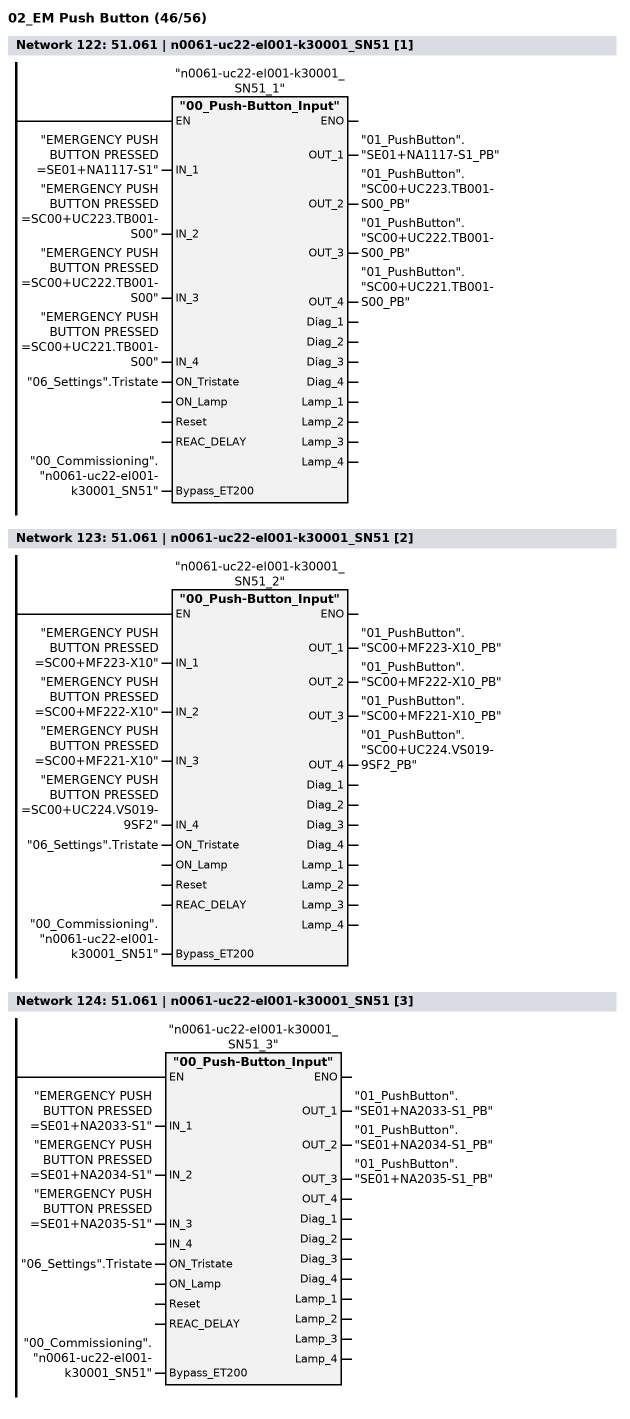
   RUNG wire#powerrail
      "n0061-uc22-el001-k30001_SN51_1"(IN_1 := "EMERGENCY PUSH BUTTON PRESSED =SE01+NA1117-S1", IN_2 := "EMERGENCY PUSH BUTTON PRESSED =SC00+UC223.TB001-S00", IN_3 := "EMERGENCY PUSH BUTTON PRESSED =SC00+UC222.TB001-S00", IN_4 := "EMERGENCY PUSH BUTTON PRESSED =SC00+UC221.TB001-S00", ON_Tristate := "06_Settings".Tristate, ON_Lamp :=, Reset :=, REAC_DELAY :=, Bypass_ET200 := "00_Commissioning"."n0061-uc22-el001-k30001_SN51", OUT_1 => "01_PushButton"."SE01+NA1117-S1_PB", OUT_2 => "01_PushButton"."SC00+UC223.TB001-S00_PB", OUT_3 => "01_PushButton"."SC00+UC222.TB001-S00_PB", OUT_4 => "01_PushButton"."SC00+UC221.TB001-S00_PB", Diag_1 =>, Diag_2 =>, Diag_3 =>, Diag_4 =>, Lamp_1 =>, Lamp_2 =>, Lamp_3 =>, Lamp_4 =>)
   END_RUNG
   // the same network as SCL:
   "n0061-uc22-el001-k30001_SN51_1"(IN_1 := "EMERGENCY PUSH BUTTON PRESSED =SE01+NA1117-S1",   // "00_Push-Button_Input"
                           IN_2 := "EMERGENCY PUSH BUTTON PRESSED =SC00+UC223.TB001-S00",
                           IN_3 := "EMERGENCY PUSH BUTTON PRESSED =SC00+UC222.TB001-S00",
                           IN_4 := "EMERGENCY PUSH BUTTON PRESSED =SC00+UC221.TB001-S00",
                           ON_Tristate := "06_Settings".Tristate,
                           Bypass_ET200 := "00_Commissioning"."n0061-uc22-el001-k30001_SN51",
                           OUT_1 => "01_PushButton"."SE01+NA1117-S1_PB",
                           OUT_2 => "01_PushButton"."SC00+UC223.TB001-S00_PB",
                           OUT_3 => "01_PushButton"."SC00+UC222.TB001-S00_PB",
                           OUT_4 => "01_PushButton"."SC00+UC221.TB001-S00_PB");
END_REGION

REGION Network 123: 51.061 | n0061-uc22-el001-k30001_SN51 [2]
   RUNG wire#powerrail
      "n0061-uc22-el001-k30001_SN51_2"(IN_1 := "EMERGENCY PUSH BUTTON PRESSED =SC00+MF223-X10", IN_2 := "EMERGENCY PUSH BUTTON PRESSED =SC00+MF222-X10", IN_3 := "EMERGENCY PUSH BUTTON PRESSED =SC00+MF221-X10", IN_4 := "EMERGENCY PUSH BUTTON PRESSED =SC00+UC224.VS019-9SF2", ON_Tristate := "06_Settings".Tristate, ON_Lamp :=, Reset :=, REAC_DELAY :=, Bypass_ET200 := "00_Commissioning"."n0061-uc22-el001-k30001_SN51", OUT_1 => "01_PushButton"."SC00+MF223-X10_PB", OUT_2 => "01_PushButton"."SC00+MF222-X10_PB", OUT_3 => "01_PushButton"."SC00+MF221-X10_PB", OUT_4 => "01_PushButton"."SC00+UC224.VS019-9SF2_PB", Diag_1 =>, Diag_2 =>, Diag_3 =>, Diag_4 =>, Lamp_1 =>, Lamp_2 =>, Lamp_3 =>, Lamp_4 =>)
   END_RUNG
   // the same network as SCL:
   "n0061-uc22-el001-k30001_SN51_2"(IN_1 := "EMERGENCY PUSH BUTTON PRESSED =SC00+MF223-X10",   // "00_Push-Button_Input"
                           IN_2 := "EMERGENCY PUSH BUTTON PRESSED =SC00+MF222-X10",
                           IN_3 := "EMERGENCY PUSH BUTTON PRESSED =SC00+MF221-X10",
                           IN_4 := "EMERGENCY PUSH BUTTON PRESSED =SC00+UC224.VS019-9SF2",
                           ON_Tristate := "06_Settings".Tristate,
                           Bypass_ET200 := "00_Commissioning"."n0061-uc22-el001-k30001_SN51",
                           OUT_1 => "01_PushButton"."SC00+MF223-X10_PB",
                           OUT_2 => "01_PushButton"."SC00+MF222-X10_PB",
                           OUT_3 => "01_PushButton"."SC00+MF221-X10_PB",
                           OUT_4 => "01_PushButton"."SC00+UC224.VS019-9SF2_PB");
END_REGION

REGION Network 124: 51.061 | n0061-uc22-el001-k30001_SN51 [3]
   RUNG wire#powerrail
      "n0061-uc22-el001-k30001_SN51_3"(IN_1 := "EMERGENCY PUSH BUTTON PRESSED =SE01+NA2033-S1", IN_2 := "EMERGENCY PUSH BUTTON PRESSED =SE01+NA2034-S1", IN_3 := "EMERGENCY PUSH BUTTON PRESSED =SE01+NA2035-S1", IN_4 :=, ON_Tristate := "06_Settings".Tristate, ON_Lamp :=, Reset :=, REAC_DELAY :=, Bypass_ET200 := "00_Commissioning"."n0061-uc22-el001-k30001_SN51", OUT_1 => "01_PushButton"."SE01+NA2033-S1_PB", OUT_2 => "01_PushButton"."SE01+NA2034-S1_PB", OUT_3 => "01_PushButton"."SE01+NA2035-S1_PB", OUT_4 =>, Diag_1 =>, Diag_2 =>, Diag_3 =>, Diag_4 =>, Lamp_1 =>, Lamp_2 =>, Lamp_3 =>, Lamp_4 =>)
   END_RUNG
   // the same network as SCL:
   "n0061-uc22-el001-k30001_SN51_3"(IN_1 := "EMERGENCY PUSH BUTTON PRESSED =SE01+NA2033-S1",   // "00_Push-Button_Input"
                           IN_2 := "EMERGENCY PUSH BUTTON PRESSED =SE01+NA2034-S1",
                           IN_3 := "EMERGENCY PUSH BUTTON PRESSED =SE01+NA2035-S1",
                           ON_Tristate := "06_Settings".Tristate,
                           Bypass_ET200 := "00_Commissioning"."n0061-uc22-el001-k30001_SN51",
                           OUT_1 => "01_PushButton"."SE01+NA2033-S1_PB",
                           OUT_2 => "01_PushButton"."SE01+NA2034-S1_PB",
                           OUT_3 => "01_PushButton"."SE01+NA2035-S1_PB");
END_REGION

REGION Network 125: 51.062 | n0062-uc224-xn10_SN51 [1]
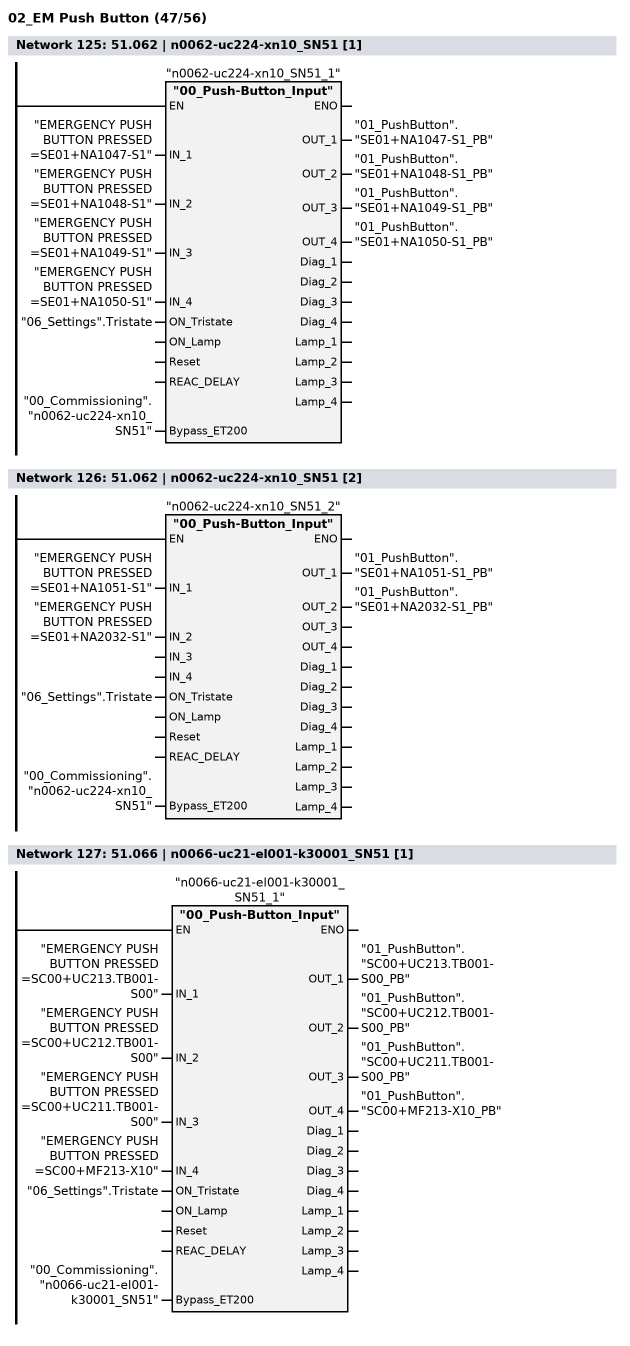
   RUNG wire#powerrail
      "n0062-uc224-xn10_SN51_1"(IN_1 := "EMERGENCY PUSH BUTTON PRESSED =SE01+NA1047-S1", IN_2 := "EMERGENCY PUSH BUTTON PRESSED =SE01+NA1048-S1", IN_3 := "EMERGENCY PUSH BUTTON PRESSED =SE01+NA1049-S1", IN_4 := "EMERGENCY PUSH BUTTON PRESSED =SE01+NA1050-S1", ON_Tristate := "06_Settings".Tristate, ON_Lamp :=, Reset :=, REAC_DELAY :=, Bypass_ET200 := "00_Commissioning"."n0062-uc224-xn10_SN51", OUT_1 => "01_PushButton"."SE01+NA1047-S1_PB", OUT_2 => "01_PushButton"."SE01+NA1048-S1_PB", OUT_3 => "01_PushButton"."SE01+NA1049-S1_PB", OUT_4 => "01_PushButton"."SE01+NA1050-S1_PB", Diag_1 =>, Diag_2 =>, Diag_3 =>, Diag_4 =>, Lamp_1 =>, Lamp_2 =>, Lamp_3 =>, Lamp_4 =>)
   END_RUNG
   // the same network as SCL:
   "n0062-uc224-xn10_SN51_1"(IN_1 := "EMERGENCY PUSH BUTTON PRESSED =SE01+NA1047-S1",   // "00_Push-Button_Input"
                           IN_2 := "EMERGENCY PUSH BUTTON PRESSED =SE01+NA1048-S1",
                           IN_3 := "EMERGENCY PUSH BUTTON PRESSED =SE01+NA1049-S1",
                           IN_4 := "EMERGENCY PUSH BUTTON PRESSED =SE01+NA1050-S1",
                           ON_Tristate := "06_Settings".Tristate,
                           Bypass_ET200 := "00_Commissioning"."n0062-uc224-xn10_SN51",
                           OUT_1 => "01_PushButton"."SE01+NA1047-S1_PB",
                           OUT_2 => "01_PushButton"."SE01+NA1048-S1_PB",
                           OUT_3 => "01_PushButton"."SE01+NA1049-S1_PB",
                           OUT_4 => "01_PushButton"."SE01+NA1050-S1_PB");
END_REGION

REGION Network 126: 51.062 | n0062-uc224-xn10_SN51 [2]
   RUNG wire#powerrail
      "n0062-uc224-xn10_SN51_2"(IN_1 := "EMERGENCY PUSH BUTTON PRESSED =SE01+NA1051-S1", IN_2 := "EMERGENCY PUSH BUTTON PRESSED =SE01+NA2032-S1", IN_3 :=, IN_4 :=, ON_Tristate := "06_Settings".Tristate, ON_Lamp :=, Reset :=, REAC_DELAY :=, Bypass_ET200 := "00_Commissioning"."n0062-uc224-xn10_SN51", OUT_1 => "01_PushButton"."SE01+NA1051-S1_PB", OUT_2 => "01_PushButton"."SE01+NA2032-S1_PB", OUT_3 =>, OUT_4 =>, Diag_1 =>, Diag_2 =>, Diag_3 =>, Diag_4 =>, Lamp_1 =>, Lamp_2 =>, Lamp_3 =>, Lamp_4 =>)
   END_RUNG
   // the same network as SCL:
   "n0062-uc224-xn10_SN51_2"(IN_1 := "EMERGENCY PUSH BUTTON PRESSED =SE01+NA1051-S1",   // "00_Push-Button_Input"
                           IN_2 := "EMERGENCY PUSH BUTTON PRESSED =SE01+NA2032-S1",
                           ON_Tristate := "06_Settings".Tristate,
                           Bypass_ET200 := "00_Commissioning"."n0062-uc224-xn10_SN51",
                           OUT_1 => "01_PushButton"."SE01+NA1051-S1_PB",
                           OUT_2 => "01_PushButton"."SE01+NA2032-S1_PB");
END_REGION

REGION Network 127: 51.066 | n0066-uc21-el001-k30001_SN51 [1]
   RUNG wire#powerrail
      "n0066-uc21-el001-k30001_SN51_1"(IN_1 := "EMERGENCY PUSH BUTTON PRESSED =SC00+UC213.TB001-S00", IN_2 := "EMERGENCY PUSH BUTTON PRESSED =SC00+UC212.TB001-S00", IN_3 := "EMERGENCY PUSH BUTTON PRESSED =SC00+UC211.TB001-S00", IN_4 := "EMERGENCY PUSH BUTTON PRESSED =SC00+MF213-X10", ON_Tristate := "06_Settings".Tristate, ON_Lamp :=, Reset :=, REAC_DELAY :=, Bypass_ET200 := "00_Commissioning"."n0066-uc21-el001-k30001_SN51", OUT_1 => "01_PushButton"."SC00+UC213.TB001-S00_PB", OUT_2 => "01_PushButton"."SC00+UC212.TB001-S00_PB", OUT_3 => "01_PushButton"."SC00+UC211.TB001-S00_PB", OUT_4 => "01_PushButton"."SC00+MF213-X10_PB", Diag_1 =>, Diag_2 =>, Diag_3 =>, Diag_4 =>, Lamp_1 =>, Lamp_2 =>, Lamp_3 =>, Lamp_4 =>)
   END_RUNG
   // the same network as SCL:
   "n0066-uc21-el001-k30001_SN51_1"(IN_1 := "EMERGENCY PUSH BUTTON PRESSED =SC00+UC213.TB001-S00",   // "00_Push-Button_Input"
                           IN_2 := "EMERGENCY PUSH BUTTON PRESSED =SC00+UC212.TB001-S00",
                           IN_3 := "EMERGENCY PUSH BUTTON PRESSED =SC00+UC211.TB001-S00",
                           IN_4 := "EMERGENCY PUSH BUTTON PRESSED =SC00+MF213-X10",
                           ON_Tristate := "06_Settings".Tristate,
                           Bypass_ET200 := "00_Commissioning"."n0066-uc21-el001-k30001_SN51",
                           OUT_1 => "01_PushButton"."SC00+UC213.TB001-S00_PB",
                           OUT_2 => "01_PushButton"."SC00+UC212.TB001-S00_PB",
                           OUT_3 => "01_PushButton"."SC00+UC211.TB001-S00_PB",
                           OUT_4 => "01_PushButton"."SC00+MF213-X10_PB");
END_REGION

REGION Network 128: 51.066 | n0066-uc21-el001-k30001_SN51 [2]
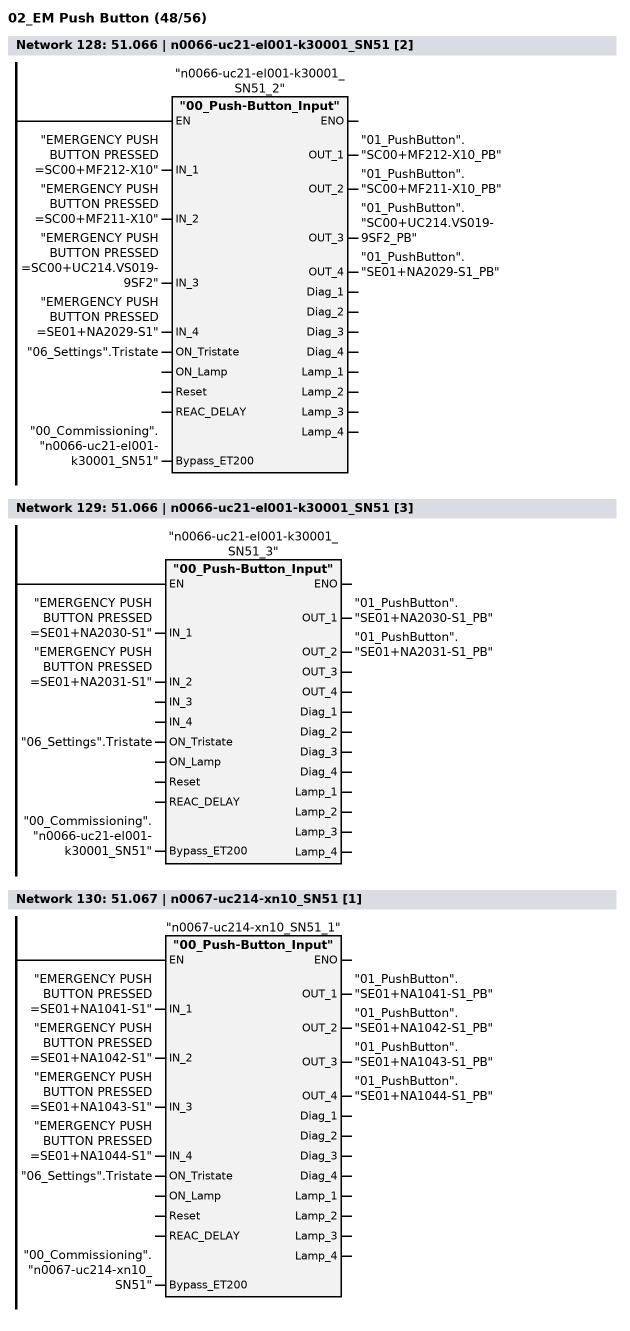
   RUNG wire#powerrail
      "n0066-uc21-el001-k30001_SN51_2"(IN_1 := "EMERGENCY PUSH BUTTON PRESSED =SC00+MF212-X10", IN_2 := "EMERGENCY PUSH BUTTON PRESSED =SC00+MF211-X10", IN_3 := "EMERGENCY PUSH BUTTON PRESSED =SC00+UC214.VS019-9SF2", IN_4 := "EMERGENCY PUSH BUTTON PRESSED =SE01+NA2029-S1", ON_Tristate := "06_Settings".Tristate, ON_Lamp :=, Reset :=, REAC_DELAY :=, Bypass_ET200 := "00_Commissioning"."n0066-uc21-el001-k30001_SN51", OUT_1 => "01_PushButton"."SC00+MF212-X10_PB", OUT_2 => "01_PushButton"."SC00+MF211-X10_PB", OUT_3 => "01_PushButton"."SC00+UC214.VS019-9SF2_PB", OUT_4 => "01_PushButton"."SE01+NA2029-S1_PB", Diag_1 =>, Diag_2 =>, Diag_3 =>, Diag_4 =>, Lamp_1 =>, Lamp_2 =>, Lamp_3 =>, Lamp_4 =>)
   END_RUNG
   // the same network as SCL:
   "n0066-uc21-el001-k30001_SN51_2"(IN_1 := "EMERGENCY PUSH BUTTON PRESSED =SC00+MF212-X10",   // "00_Push-Button_Input"
                           IN_2 := "EMERGENCY PUSH BUTTON PRESSED =SC00+MF211-X10",
                           IN_3 := "EMERGENCY PUSH BUTTON PRESSED =SC00+UC214.VS019-9SF2",
                           IN_4 := "EMERGENCY PUSH BUTTON PRESSED =SE01+NA2029-S1",
                           ON_Tristate := "06_Settings".Tristate,
                           Bypass_ET200 := "00_Commissioning"."n0066-uc21-el001-k30001_SN51",
                           OUT_1 => "01_PushButton"."SC00+MF212-X10_PB",
                           OUT_2 => "01_PushButton"."SC00+MF211-X10_PB",
                           OUT_3 => "01_PushButton"."SC00+UC214.VS019-9SF2_PB",
                           OUT_4 => "01_PushButton"."SE01+NA2029-S1_PB");
END_REGION

REGION Network 129: 51.066 | n0066-uc21-el001-k30001_SN51 [3]
   RUNG wire#powerrail
      "n0066-uc21-el001-k30001_SN51_3"(IN_1 := "EMERGENCY PUSH BUTTON PRESSED =SE01+NA2030-S1", IN_2 := "EMERGENCY PUSH BUTTON PRESSED =SE01+NA2031-S1", IN_3 :=, IN_4 :=, ON_Tristate := "06_Settings".Tristate, ON_Lamp :=, Reset :=, REAC_DELAY :=, Bypass_ET200 := "00_Commissioning"."n0066-uc21-el001-k30001_SN51", OUT_1 => "01_PushButton"."SE01+NA2030-S1_PB", OUT_2 => "01_PushButton"."SE01+NA2031-S1_PB", OUT_3 =>, OUT_4 =>, Diag_1 =>, Diag_2 =>, Diag_3 =>, Diag_4 =>, Lamp_1 =>, Lamp_2 =>, Lamp_3 =>, Lamp_4 =>)
   END_RUNG
   // the same network as SCL:
   "n0066-uc21-el001-k30001_SN51_3"(IN_1 := "EMERGENCY PUSH BUTTON PRESSED =SE01+NA2030-S1",   // "00_Push-Button_Input"
                           IN_2 := "EMERGENCY PUSH BUTTON PRESSED =SE01+NA2031-S1",
                           ON_Tristate := "06_Settings".Tristate,
                           Bypass_ET200 := "00_Commissioning"."n0066-uc21-el001-k30001_SN51",
                           OUT_1 => "01_PushButton"."SE01+NA2030-S1_PB",
                           OUT_2 => "01_PushButton"."SE01+NA2031-S1_PB");
END_REGION

REGION Network 130: 51.067 | n0067-uc214-xn10_SN51 [1]
   RUNG wire#powerrail
      "n0067-uc214-xn10_SN51_1"(IN_1 := "EMERGENCY PUSH BUTTON PRESSED =SE01+NA1041-S1", IN_2 := "EMERGENCY PUSH BUTTON PRESSED =SE01+NA1042-S1", IN_3 := "EMERGENCY PUSH BUTTON PRESSED =SE01+NA1043-S1", IN_4 := "EMERGENCY PUSH BUTTON PRESSED =SE01+NA1044-S1", ON_Tristate := "06_Settings".Tristate, ON_Lamp :=, Reset :=, REAC_DELAY :=, Bypass_ET200 := "00_Commissioning"."n0067-uc214-xn10_SN51", OUT_1 => "01_PushButton"."SE01+NA1041-S1_PB", OUT_2 => "01_PushButton"."SE01+NA1042-S1_PB", OUT_3 => "01_PushButton"."SE01+NA1043-S1_PB", OUT_4 => "01_PushButton"."SE01+NA1044-S1_PB", Diag_1 =>, Diag_2 =>, Diag_3 =>, Diag_4 =>, Lamp_1 =>, Lamp_2 =>, Lamp_3 =>, Lamp_4 =>)
   END_RUNG
   // the same network as SCL:
   "n0067-uc214-xn10_SN51_1"(IN_1 := "EMERGENCY PUSH BUTTON PRESSED =SE01+NA1041-S1",   // "00_Push-Button_Input"
                           IN_2 := "EMERGENCY PUSH BUTTON PRESSED =SE01+NA1042-S1",
                           IN_3 := "EMERGENCY PUSH BUTTON PRESSED =SE01+NA1043-S1",
                           IN_4 := "EMERGENCY PUSH BUTTON PRESSED =SE01+NA1044-S1",
                           ON_Tristate := "06_Settings".Tristate,
                           Bypass_ET200 := "00_Commissioning"."n0067-uc214-xn10_SN51",
                           OUT_1 => "01_PushButton"."SE01+NA1041-S1_PB",
                           OUT_2 => "01_PushButton"."SE01+NA1042-S1_PB",
                           OUT_3 => "01_PushButton"."SE01+NA1043-S1_PB",
                           OUT_4 => "01_PushButton"."SE01+NA1044-S1_PB");
END_REGION

REGION Network 131: 51.067 | n0067-uc214-xn10_SN51 [2]
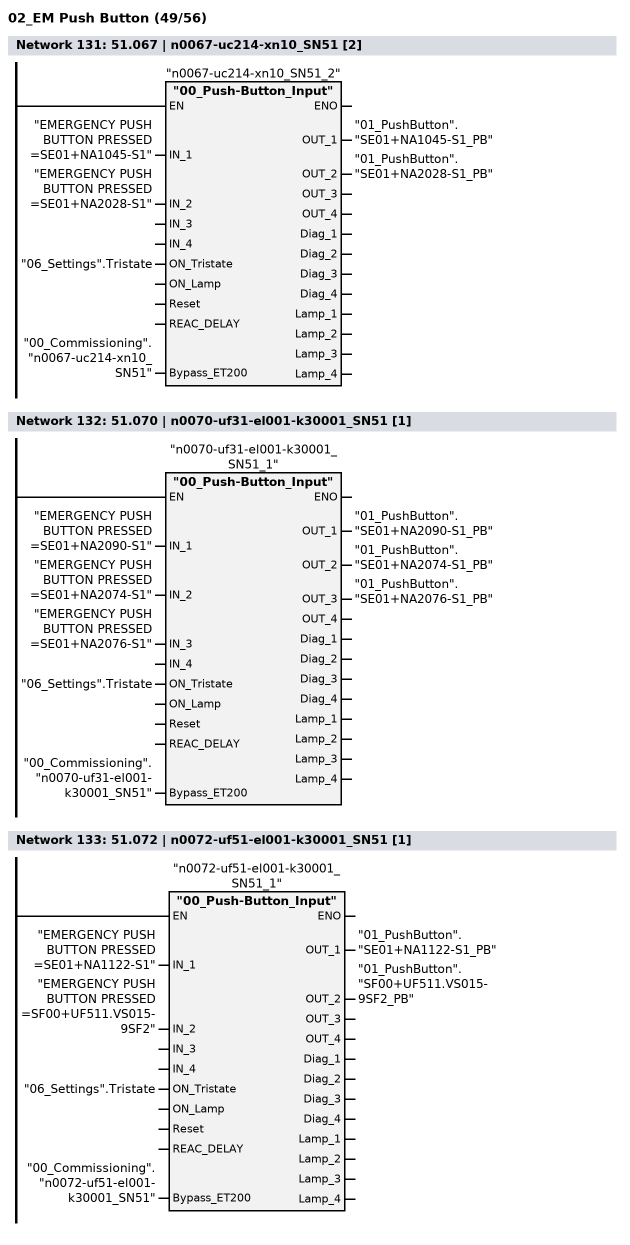
   RUNG wire#powerrail
      "n0067-uc214-xn10_SN51_2"(IN_1 := "EMERGENCY PUSH BUTTON PRESSED =SE01+NA1045-S1", IN_2 := "EMERGENCY PUSH BUTTON PRESSED =SE01+NA2028-S1", IN_3 :=, IN_4 :=, ON_Tristate := "06_Settings".Tristate, ON_Lamp :=, Reset :=, REAC_DELAY :=, Bypass_ET200 := "00_Commissioning"."n0067-uc214-xn10_SN51", OUT_1 => "01_PushButton"."SE01+NA1045-S1_PB", OUT_2 => "01_PushButton"."SE01+NA2028-S1_PB", OUT_3 =>, OUT_4 =>, Diag_1 =>, Diag_2 =>, Diag_3 =>, Diag_4 =>, Lamp_1 =>, Lamp_2 =>, Lamp_3 =>, Lamp_4 =>)
   END_RUNG
   // the same network as SCL:
   "n0067-uc214-xn10_SN51_2"(IN_1 := "EMERGENCY PUSH BUTTON PRESSED =SE01+NA1045-S1",   // "00_Push-Button_Input"
                           IN_2 := "EMERGENCY PUSH BUTTON PRESSED =SE01+NA2028-S1",
                           ON_Tristate := "06_Settings".Tristate,
                           Bypass_ET200 := "00_Commissioning"."n0067-uc214-xn10_SN51",
                           OUT_1 => "01_PushButton"."SE01+NA1045-S1_PB",
                           OUT_2 => "01_PushButton"."SE01+NA2028-S1_PB");
END_REGION

REGION Network 132: 51.070 | n0070-uf31-el001-k30001_SN51 [1]
   RUNG wire#powerrail
      "n0070-uf31-el001-k30001_SN51_1"(IN_1 := "EMERGENCY PUSH BUTTON PRESSED =SE01+NA2090-S1", IN_2 := "EMERGENCY PUSH BUTTON PRESSED =SE01+NA2074-S1", IN_3 := "EMERGENCY PUSH BUTTON PRESSED =SE01+NA2076-S1", IN_4 :=, ON_Tristate := "06_Settings".Tristate, ON_Lamp :=, Reset :=, REAC_DELAY :=, Bypass_ET200 := "00_Commissioning"."n0070-uf31-el001-k30001_SN51", OUT_1 => "01_PushButton"."SE01+NA2090-S1_PB", OUT_2 => "01_PushButton"."SE01+NA2074-S1_PB", OUT_3 => "01_PushButton"."SE01+NA2076-S1_PB", OUT_4 =>, Diag_1 =>, Diag_2 =>, Diag_3 =>, Diag_4 =>, Lamp_1 =>, Lamp_2 =>, Lamp_3 =>, Lamp_4 =>)
   END_RUNG
   // the same network as SCL:
   "n0070-uf31-el001-k30001_SN51_1"(IN_1 := "EMERGENCY PUSH BUTTON PRESSED =SE01+NA2090-S1",   // "00_Push-Button_Input"
                           IN_2 := "EMERGENCY PUSH BUTTON PRESSED =SE01+NA2074-S1",
                           IN_3 := "EMERGENCY PUSH BUTTON PRESSED =SE01+NA2076-S1",
                           ON_Tristate := "06_Settings".Tristate,
                           Bypass_ET200 := "00_Commissioning"."n0070-uf31-el001-k30001_SN51",
                           OUT_1 => "01_PushButton"."SE01+NA2090-S1_PB",
                           OUT_2 => "01_PushButton"."SE01+NA2074-S1_PB",
                           OUT_3 => "01_PushButton"."SE01+NA2076-S1_PB");
END_REGION

REGION Network 133: 51.072 | n0072-uf51-el001-k30001_SN51 [1]
   RUNG wire#powerrail
      "n0072-uf51-el001-k30001_SN51_1"(IN_1 := "EMERGENCY PUSH BUTTON PRESSED =SE01+NA1122-S1", IN_2 := "EMERGENCY PUSH BUTTON PRESSED =SF00+UF511.VS015-9SF2", IN_3 :=, IN_4 :=, ON_Tristate := "06_Settings".Tristate, ON_Lamp :=, Reset :=, REAC_DELAY :=, Bypass_ET200 := "00_Commissioning"."n0072-uf51-el001-k30001_SN51", OUT_1 => "01_PushButton"."SE01+NA1122-S1_PB", OUT_2 => "01_PushButton"."SF00+UF511.VS015-9SF2_PB", OUT_3 =>, OUT_4 =>, Diag_1 =>, Diag_2 =>, Diag_3 =>, Diag_4 =>, Lamp_1 =>, Lamp_2 =>, Lamp_3 =>, Lamp_4 =>)
   END_RUNG
   // the same network as SCL:
   "n0072-uf51-el001-k30001_SN51_1"(IN_1 := "EMERGENCY PUSH BUTTON PRESSED =SE01+NA1122-S1",   // "00_Push-Button_Input"
                           IN_2 := "EMERGENCY PUSH BUTTON PRESSED =SF00+UF511.VS015-9SF2",
                           ON_Tristate := "06_Settings".Tristate,
                           Bypass_ET200 := "00_Commissioning"."n0072-uf51-el001-k30001_SN51",
                           OUT_1 => "01_PushButton"."SE01+NA1122-S1_PB",
                           OUT_2 => "01_PushButton"."SF00+UF511.VS015-9SF2_PB");
END_REGION

REGION Network 134: 51.080 | n0080-uf511-xn10_SN51 [1]
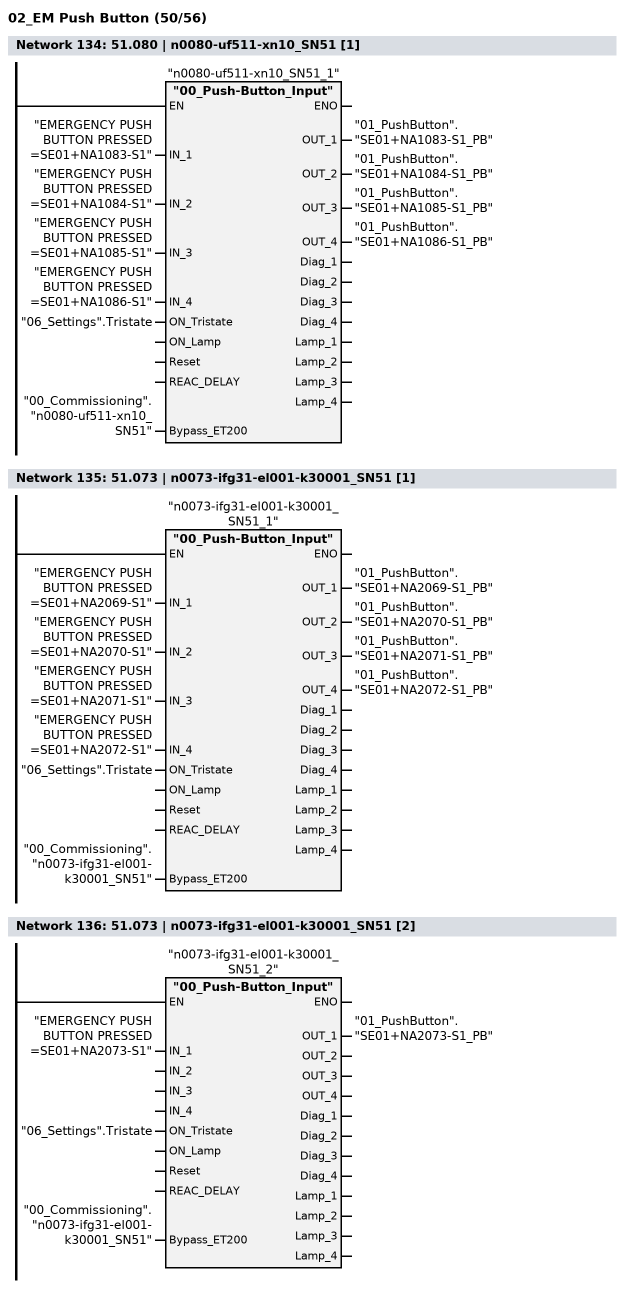
   RUNG wire#powerrail
      "n0080-uf511-xn10_SN51_1"(IN_1 := "EMERGENCY PUSH BUTTON PRESSED =SE01+NA1083-S1", IN_2 := "EMERGENCY PUSH BUTTON PRESSED =SE01+NA1084-S1", IN_3 := "EMERGENCY PUSH BUTTON PRESSED =SE01+NA1085-S1", IN_4 := "EMERGENCY PUSH BUTTON PRESSED =SE01+NA1086-S1", ON_Tristate := "06_Settings".Tristate, ON_Lamp :=, Reset :=, REAC_DELAY :=, Bypass_ET200 := "00_Commissioning"."n0080-uf511-xn10_SN51", OUT_1 => "01_PushButton"."SE01+NA1083-S1_PB", OUT_2 => "01_PushButton"."SE01+NA1084-S1_PB", OUT_3 => "01_PushButton"."SE01+NA1085-S1_PB", OUT_4 => "01_PushButton"."SE01+NA1086-S1_PB", Diag_1 =>, Diag_2 =>, Diag_3 =>, Diag_4 =>, Lamp_1 =>, Lamp_2 =>, Lamp_3 =>, Lamp_4 =>)
   END_RUNG
   // the same network as SCL:
   "n0080-uf511-xn10_SN51_1"(IN_1 := "EMERGENCY PUSH BUTTON PRESSED =SE01+NA1083-S1",   // "00_Push-Button_Input"
                           IN_2 := "EMERGENCY PUSH BUTTON PRESSED =SE01+NA1084-S1",
                           IN_3 := "EMERGENCY PUSH BUTTON PRESSED =SE01+NA1085-S1",
                           IN_4 := "EMERGENCY PUSH BUTTON PRESSED =SE01+NA1086-S1",
                           ON_Tristate := "06_Settings".Tristate,
                           Bypass_ET200 := "00_Commissioning"."n0080-uf511-xn10_SN51",
                           OUT_1 => "01_PushButton"."SE01+NA1083-S1_PB",
                           OUT_2 => "01_PushButton"."SE01+NA1084-S1_PB",
                           OUT_3 => "01_PushButton"."SE01+NA1085-S1_PB",
                           OUT_4 => "01_PushButton"."SE01+NA1086-S1_PB");
END_REGION

REGION Network 135: 51.073 | n0073-ifg31-el001-k30001_SN51 [1]
   RUNG wire#powerrail
      "n0073-ifg31-el001-k30001_SN51_1"(IN_1 := "EMERGENCY PUSH BUTTON PRESSED =SE01+NA2069-S1", IN_2 := "EMERGENCY PUSH BUTTON PRESSED =SE01+NA2070-S1", IN_3 := "EMERGENCY PUSH BUTTON PRESSED =SE01+NA2071-S1", IN_4 := "EMERGENCY PUSH BUTTON PRESSED =SE01+NA2072-S1", ON_Tristate := "06_Settings".Tristate, ON_Lamp :=, Reset :=, REAC_DELAY :=, Bypass_ET200 := "00_Commissioning"."n0073-ifg31-el001-k30001_SN51", OUT_1 => "01_PushButton"."SE01+NA2069-S1_PB", OUT_2 => "01_PushButton"."SE01+NA2070-S1_PB", OUT_3 => "01_PushButton"."SE01+NA2071-S1_PB", OUT_4 => "01_PushButton"."SE01+NA2072-S1_PB", Diag_1 =>, Diag_2 =>, Diag_3 =>, Diag_4 =>, Lamp_1 =>, Lamp_2 =>, Lamp_3 =>, Lamp_4 =>)
   END_RUNG
   // the same network as SCL:
   "n0073-ifg31-el001-k30001_SN51_1"(IN_1 := "EMERGENCY PUSH BUTTON PRESSED =SE01+NA2069-S1",   // "00_Push-Button_Input"
                           IN_2 := "EMERGENCY PUSH BUTTON PRESSED =SE01+NA2070-S1",
                           IN_3 := "EMERGENCY PUSH BUTTON PRESSED =SE01+NA2071-S1",
                           IN_4 := "EMERGENCY PUSH BUTTON PRESSED =SE01+NA2072-S1",
                           ON_Tristate := "06_Settings".Tristate,
                           Bypass_ET200 := "00_Commissioning"."n0073-ifg31-el001-k30001_SN51",
                           OUT_1 => "01_PushButton"."SE01+NA2069-S1_PB",
                           OUT_2 => "01_PushButton"."SE01+NA2070-S1_PB",
                           OUT_3 => "01_PushButton"."SE01+NA2071-S1_PB",
                           OUT_4 => "01_PushButton"."SE01+NA2072-S1_PB");
END_REGION

REGION Network 136: 51.073 | n0073-ifg31-el001-k30001_SN51 [2]
   RUNG wire#powerrail
      "n0073-ifg31-el001-k30001_SN51_2"(IN_1 := "EMERGENCY PUSH BUTTON PRESSED =SE01+NA2073-S1", IN_2 :=, IN_3 :=, IN_4 :=, ON_Tristate := "06_Settings".Tristate, ON_Lamp :=, Reset :=, REAC_DELAY :=, Bypass_ET200 := "00_Commissioning"."n0073-ifg31-el001-k30001_SN51", OUT_1 => "01_PushButton"."SE01+NA2073-S1_PB", OUT_2 =>, OUT_3 =>, OUT_4 =>, Diag_1 =>, Diag_2 =>, Diag_3 =>, Diag_4 =>, Lamp_1 =>, Lamp_2 =>, Lamp_3 =>, Lamp_4 =>)
   END_RUNG
   // the same network as SCL:
   "n0073-ifg31-el001-k30001_SN51_2"(IN_1 := "EMERGENCY PUSH BUTTON PRESSED =SE01+NA2073-S1",   // "00_Push-Button_Input"
                           ON_Tristate := "06_Settings".Tristate,
                           Bypass_ET200 := "00_Commissioning"."n0073-ifg31-el001-k30001_SN51",
                           OUT_1 => "01_PushButton"."SE01+NA2073-S1_PB");
END_REGION

REGION Network 137: 51.074 | n0074-ifg41-el001-k30001_SN51 [1]
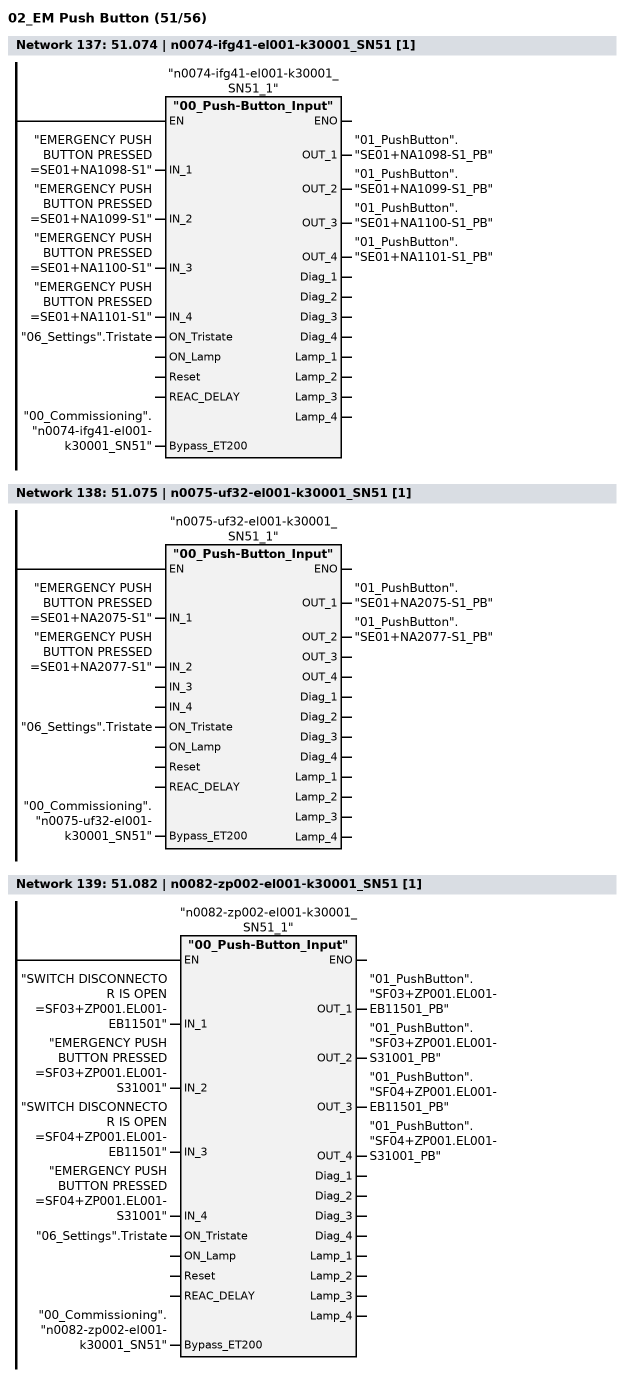
   RUNG wire#powerrail
      "n0074-ifg41-el001-k30001_SN51_1"(IN_1 := "EMERGENCY PUSH BUTTON PRESSED =SE01+NA1098-S1", IN_2 := "EMERGENCY PUSH BUTTON PRESSED =SE01+NA1099-S1", IN_3 := "EMERGENCY PUSH BUTTON PRESSED =SE01+NA1100-S1", IN_4 := "EMERGENCY PUSH BUTTON PRESSED =SE01+NA1101-S1", ON_Tristate := "06_Settings".Tristate, ON_Lamp :=, Reset :=, REAC_DELAY :=, Bypass_ET200 := "00_Commissioning"."n0074-ifg41-el001-k30001_SN51", OUT_1 => "01_PushButton"."SE01+NA1098-S1_PB", OUT_2 => "01_PushButton"."SE01+NA1099-S1_PB", OUT_3 => "01_PushButton"."SE01+NA1100-S1_PB", OUT_4 => "01_PushButton"."SE01+NA1101-S1_PB", Diag_1 =>, Diag_2 =>, Diag_3 =>, Diag_4 =>, Lamp_1 =>, Lamp_2 =>, Lamp_3 =>, Lamp_4 =>)
   END_RUNG
   // the same network as SCL:
   "n0074-ifg41-el001-k30001_SN51_1"(IN_1 := "EMERGENCY PUSH BUTTON PRESSED =SE01+NA1098-S1",   // "00_Push-Button_Input"
                           IN_2 := "EMERGENCY PUSH BUTTON PRESSED =SE01+NA1099-S1",
                           IN_3 := "EMERGENCY PUSH BUTTON PRESSED =SE01+NA1100-S1",
                           IN_4 := "EMERGENCY PUSH BUTTON PRESSED =SE01+NA1101-S1",
                           ON_Tristate := "06_Settings".Tristate,
                           Bypass_ET200 := "00_Commissioning"."n0074-ifg41-el001-k30001_SN51",
                           OUT_1 => "01_PushButton"."SE01+NA1098-S1_PB",
                           OUT_2 => "01_PushButton"."SE01+NA1099-S1_PB",
                           OUT_3 => "01_PushButton"."SE01+NA1100-S1_PB",
                           OUT_4 => "01_PushButton"."SE01+NA1101-S1_PB");
END_REGION

REGION Network 138: 51.075 | n0075-uf32-el001-k30001_SN51 [1]
   RUNG wire#powerrail
      "n0075-uf32-el001-k30001_SN51_1"(IN_1 := "EMERGENCY PUSH BUTTON PRESSED =SE01+NA2075-S1", IN_2 := "EMERGENCY PUSH BUTTON PRESSED =SE01+NA2077-S1", IN_3 :=, IN_4 :=, ON_Tristate := "06_Settings".Tristate, ON_Lamp :=, Reset :=, REAC_DELAY :=, Bypass_ET200 := "00_Commissioning"."n0075-uf32-el001-k30001_SN51", OUT_1 => "01_PushButton"."SE01+NA2075-S1_PB", OUT_2 => "01_PushButton"."SE01+NA2077-S1_PB", OUT_3 =>, OUT_4 =>, Diag_1 =>, Diag_2 =>, Diag_3 =>, Diag_4 =>, Lamp_1 =>, Lamp_2 =>, Lamp_3 =>, Lamp_4 =>)
   END_RUNG
   // the same network as SCL:
   "n0075-uf32-el001-k30001_SN51_1"(IN_1 := "EMERGENCY PUSH BUTTON PRESSED =SE01+NA2075-S1",   // "00_Push-Button_Input"
                           IN_2 := "EMERGENCY PUSH BUTTON PRESSED =SE01+NA2077-S1",
                           ON_Tristate := "06_Settings".Tristate,
                           Bypass_ET200 := "00_Commissioning"."n0075-uf32-el001-k30001_SN51",
                           OUT_1 => "01_PushButton"."SE01+NA2075-S1_PB",
                           OUT_2 => "01_PushButton"."SE01+NA2077-S1_PB");
END_REGION

REGION Network 139: 51.082 | n0082-zp002-el001-k30001_SN51 [1]
   RUNG wire#powerrail
      "n0082-zp002-el001-k30001_SN51_1"(IN_1 := "SWITCH DISCONNECTOR IS OPEN =SF03+ZP001.EL001-EB11501", IN_2 := "EMERGENCY PUSH BUTTON PRESSED =SF03+ZP001.EL001-S31001", IN_3 := "SWITCH DISCONNECTOR IS OPEN =SF04+ZP001.EL001-EB11501", IN_4 := "EMERGENCY PUSH BUTTON PRESSED =SF04+ZP001.EL001-S31001", ON_Tristate := "06_Settings".Tristate, ON_Lamp :=, Reset :=, REAC_DELAY :=, Bypass_ET200 := "00_Commissioning"."n0082-zp002-el001-k30001_SN51", OUT_1 => "01_PushButton"."SF03+ZP001.EL001-EB11501_PB", OUT_2 => "01_PushButton"."SF03+ZP001.EL001-S31001_PB", OUT_3 => "01_PushButton"."SF04+ZP001.EL001-EB11501_PB", OUT_4 => "01_PushButton"."SF04+ZP001.EL001-S31001_PB", Diag_1 =>, Diag_2 =>, Diag_3 =>, Diag_4 =>, Lamp_1 =>, Lamp_2 =>, Lamp_3 =>, Lamp_4 =>)
   END_RUNG
   // the same network as SCL:
   "n0082-zp002-el001-k30001_SN51_1"(IN_1 := "SWITCH DISCONNECTOR IS OPEN =SF03+ZP001.EL001-EB11501",   // "00_Push-Button_Input"
                           IN_2 := "EMERGENCY PUSH BUTTON PRESSED =SF03+ZP001.EL001-S31001",
                           IN_3 := "SWITCH DISCONNECTOR IS OPEN =SF04+ZP001.EL001-EB11501",
                           IN_4 := "EMERGENCY PUSH BUTTON PRESSED =SF04+ZP001.EL001-S31001",
                           ON_Tristate := "06_Settings".Tristate,
                           Bypass_ET200 := "00_Commissioning"."n0082-zp002-el001-k30001_SN51",
                           OUT_1 => "01_PushButton"."SF03+ZP001.EL001-EB11501_PB",
                           OUT_2 => "01_PushButton"."SF03+ZP001.EL001-S31001_PB",
                           OUT_3 => "01_PushButton"."SF04+ZP001.EL001-EB11501_PB",
                           OUT_4 => "01_PushButton"."SF04+ZP001.EL001-S31001_PB");
END_REGION

REGION Network 140: 51.083 | n0083-lv001-el001-k30001_SN51 [1]
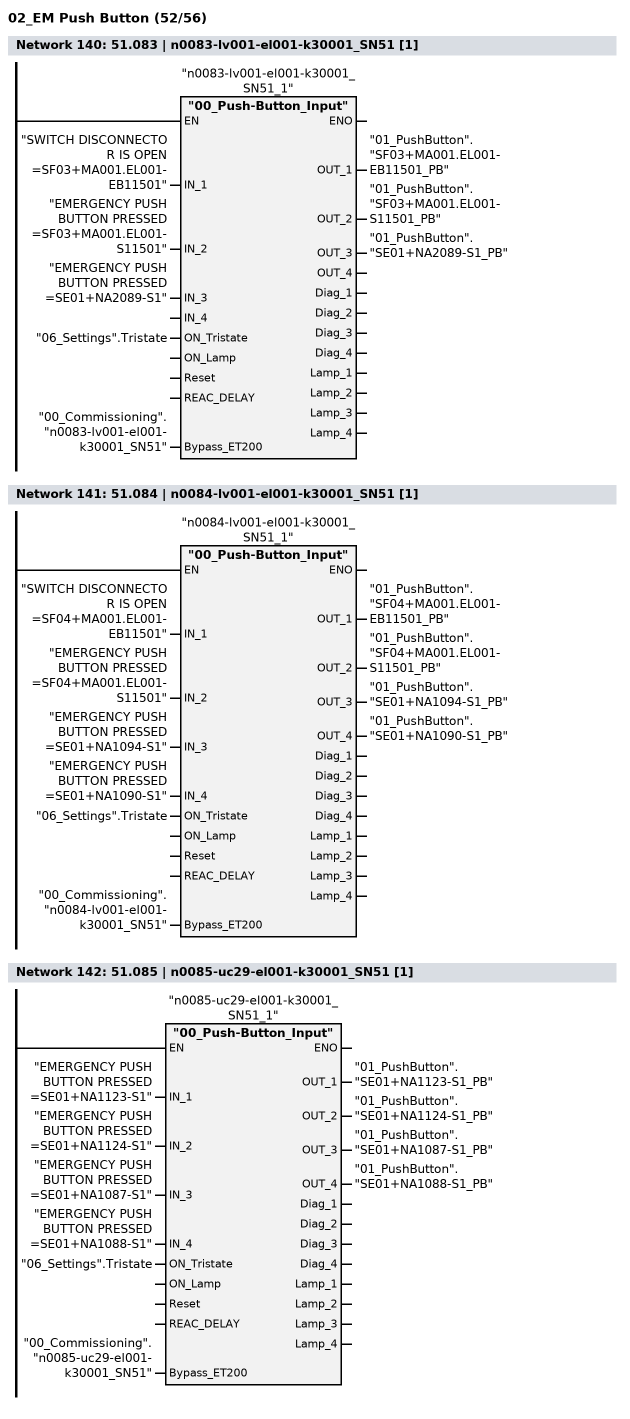
   RUNG wire#powerrail
      "n0083-lv001-el001-k30001_SN51_1"(IN_1 := "SWITCH DISCONNECTOR IS OPEN =SF03+MA001.EL001-EB11501", IN_2 := "EMERGENCY PUSH BUTTON PRESSED =SF03+MA001.EL001-S11501", IN_3 := "EMERGENCY PUSH BUTTON PRESSED =SE01+NA2089-S1", IN_4 :=, ON_Tristate := "06_Settings".Tristate, ON_Lamp :=, Reset :=, REAC_DELAY :=, Bypass_ET200 := "00_Commissioning"."n0083-lv001-el001-k30001_SN51", OUT_1 => "01_PushButton"."SF03+MA001.EL001-EB11501_PB", OUT_2 => "01_PushButton"."SF03+MA001.EL001-S11501_PB", OUT_3 => "01_PushButton"."SE01+NA2089-S1_PB", OUT_4 =>, Diag_1 =>, Diag_2 =>, Diag_3 =>, Diag_4 =>, Lamp_1 =>, Lamp_2 =>, Lamp_3 =>, Lamp_4 =>)
   END_RUNG
   // the same network as SCL:
   "n0083-lv001-el001-k30001_SN51_1"(IN_1 := "SWITCH DISCONNECTOR IS OPEN =SF03+MA001.EL001-EB11501",   // "00_Push-Button_Input"
                           IN_2 := "EMERGENCY PUSH BUTTON PRESSED =SF03+MA001.EL001-S11501",
                           IN_3 := "EMERGENCY PUSH BUTTON PRESSED =SE01+NA2089-S1",
                           ON_Tristate := "06_Settings".Tristate,
                           Bypass_ET200 := "00_Commissioning"."n0083-lv001-el001-k30001_SN51",
                           OUT_1 => "01_PushButton"."SF03+MA001.EL001-EB11501_PB",
                           OUT_2 => "01_PushButton"."SF03+MA001.EL001-S11501_PB",
                           OUT_3 => "01_PushButton"."SE01+NA2089-S1_PB");
END_REGION

REGION Network 141: 51.084 | n0084-lv001-el001-k30001_SN51 [1]
   RUNG wire#powerrail
      "n0084-lv001-el001-k30001_SN51_1"(IN_1 := "SWITCH DISCONNECTOR IS OPEN =SF04+MA001.EL001-EB11501", IN_2 := "EMERGENCY PUSH BUTTON PRESSED =SF04+MA001.EL001-S11501", IN_3 := "EMERGENCY PUSH BUTTON PRESSED =SE01+NA1094-S1", IN_4 := "EMERGENCY PUSH BUTTON PRESSED =SE01+NA1090-S1", ON_Tristate := "06_Settings".Tristate, ON_Lamp :=, Reset :=, REAC_DELAY :=, Bypass_ET200 := "00_Commissioning"."n0084-lv001-el001-k30001_SN51", OUT_1 => "01_PushButton"."SF04+MA001.EL001-EB11501_PB", OUT_2 => "01_PushButton"."SF04+MA001.EL001-S11501_PB", OUT_3 => "01_PushButton"."SE01+NA1094-S1_PB", OUT_4 => "01_PushButton"."SE01+NA1090-S1_PB", Diag_1 =>, Diag_2 =>, Diag_3 =>, Diag_4 =>, Lamp_1 =>, Lamp_2 =>, Lamp_3 =>, Lamp_4 =>)
   END_RUNG
   // the same network as SCL:
   "n0084-lv001-el001-k30001_SN51_1"(IN_1 := "SWITCH DISCONNECTOR IS OPEN =SF04+MA001.EL001-EB11501",   // "00_Push-Button_Input"
                           IN_2 := "EMERGENCY PUSH BUTTON PRESSED =SF04+MA001.EL001-S11501",
                           IN_3 := "EMERGENCY PUSH BUTTON PRESSED =SE01+NA1094-S1",
                           IN_4 := "EMERGENCY PUSH BUTTON PRESSED =SE01+NA1090-S1",
                           ON_Tristate := "06_Settings".Tristate,
                           Bypass_ET200 := "00_Commissioning"."n0084-lv001-el001-k30001_SN51",
                           OUT_1 => "01_PushButton"."SF04+MA001.EL001-EB11501_PB",
                           OUT_2 => "01_PushButton"."SF04+MA001.EL001-S11501_PB",
                           OUT_3 => "01_PushButton"."SE01+NA1094-S1_PB",
                           OUT_4 => "01_PushButton"."SE01+NA1090-S1_PB");
END_REGION

REGION Network 142: 51.085 | n0085-uc29-el001-k30001_SN51 [1]
   RUNG wire#powerrail
      "n0085-uc29-el001-k30001_SN51_1"(IN_1 := "EMERGENCY PUSH BUTTON PRESSED =SE01+NA1123-S1", IN_2 := "EMERGENCY PUSH BUTTON PRESSED =SE01+NA1124-S1", IN_3 := "EMERGENCY PUSH BUTTON PRESSED =SE01+NA1087-S1", IN_4 := "EMERGENCY PUSH BUTTON PRESSED =SE01+NA1088-S1", ON_Tristate := "06_Settings".Tristate, ON_Lamp :=, Reset :=, REAC_DELAY :=, Bypass_ET200 := "00_Commissioning"."n0085-uc29-el001-k30001_SN51", OUT_1 => "01_PushButton"."SE01+NA1123-S1_PB", OUT_2 => "01_PushButton"."SE01+NA1124-S1_PB", OUT_3 => "01_PushButton"."SE01+NA1087-S1_PB", OUT_4 => "01_PushButton"."SE01+NA1088-S1_PB", Diag_1 =>, Diag_2 =>, Diag_3 =>, Diag_4 =>, Lamp_1 =>, Lamp_2 =>, Lamp_3 =>, Lamp_4 =>)
   END_RUNG
   // the same network as SCL:
   "n0085-uc29-el001-k30001_SN51_1"(IN_1 := "EMERGENCY PUSH BUTTON PRESSED =SE01+NA1123-S1",   // "00_Push-Button_Input"
                           IN_2 := "EMERGENCY PUSH BUTTON PRESSED =SE01+NA1124-S1",
                           IN_3 := "EMERGENCY PUSH BUTTON PRESSED =SE01+NA1087-S1",
                           IN_4 := "EMERGENCY PUSH BUTTON PRESSED =SE01+NA1088-S1",
                           ON_Tristate := "06_Settings".Tristate,
                           Bypass_ET200 := "00_Commissioning"."n0085-uc29-el001-k30001_SN51",
                           OUT_1 => "01_PushButton"."SE01+NA1123-S1_PB",
                           OUT_2 => "01_PushButton"."SE01+NA1124-S1_PB",
                           OUT_3 => "01_PushButton"."SE01+NA1087-S1_PB",
                           OUT_4 => "01_PushButton"."SE01+NA1088-S1_PB");
END_REGION

REGION Network 143: 51.085 | n0085-uc29-el001-k30001_SN51 [2]
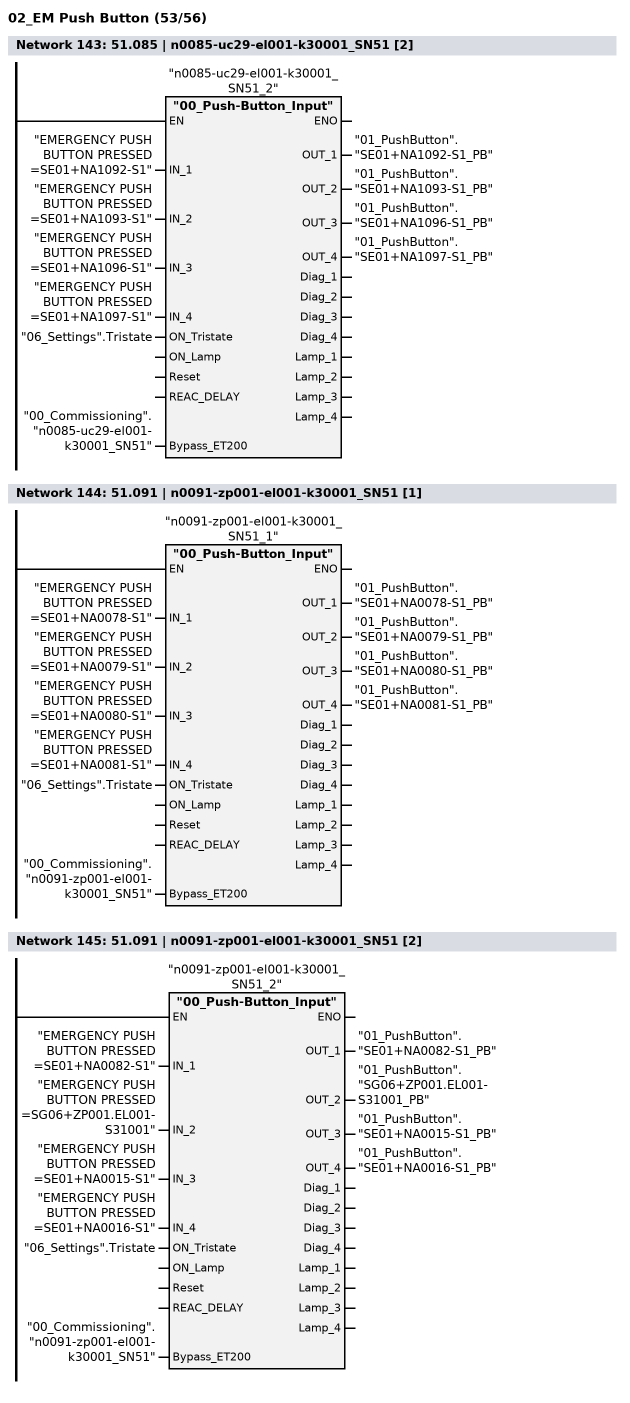
   RUNG wire#powerrail
      "n0085-uc29-el001-k30001_SN51_2"(IN_1 := "EMERGENCY PUSH BUTTON PRESSED =SE01+NA1092-S1", IN_2 := "EMERGENCY PUSH BUTTON PRESSED =SE01+NA1093-S1", IN_3 := "EMERGENCY PUSH BUTTON PRESSED =SE01+NA1096-S1", IN_4 := "EMERGENCY PUSH BUTTON PRESSED =SE01+NA1097-S1", ON_Tristate := "06_Settings".Tristate, ON_Lamp :=, Reset :=, REAC_DELAY :=, Bypass_ET200 := "00_Commissioning"."n0085-uc29-el001-k30001_SN51", OUT_1 => "01_PushButton"."SE01+NA1092-S1_PB", OUT_2 => "01_PushButton"."SE01+NA1093-S1_PB", OUT_3 => "01_PushButton"."SE01+NA1096-S1_PB", OUT_4 => "01_PushButton"."SE01+NA1097-S1_PB", Diag_1 =>, Diag_2 =>, Diag_3 =>, Diag_4 =>, Lamp_1 =>, Lamp_2 =>, Lamp_3 =>, Lamp_4 =>)
   END_RUNG
   // the same network as SCL:
   "n0085-uc29-el001-k30001_SN51_2"(IN_1 := "EMERGENCY PUSH BUTTON PRESSED =SE01+NA1092-S1",   // "00_Push-Button_Input"
                           IN_2 := "EMERGENCY PUSH BUTTON PRESSED =SE01+NA1093-S1",
                           IN_3 := "EMERGENCY PUSH BUTTON PRESSED =SE01+NA1096-S1",
                           IN_4 := "EMERGENCY PUSH BUTTON PRESSED =SE01+NA1097-S1",
                           ON_Tristate := "06_Settings".Tristate,
                           Bypass_ET200 := "00_Commissioning"."n0085-uc29-el001-k30001_SN51",
                           OUT_1 => "01_PushButton"."SE01+NA1092-S1_PB",
                           OUT_2 => "01_PushButton"."SE01+NA1093-S1_PB",
                           OUT_3 => "01_PushButton"."SE01+NA1096-S1_PB",
                           OUT_4 => "01_PushButton"."SE01+NA1097-S1_PB");
END_REGION

REGION Network 144: 51.091 | n0091-zp001-el001-k30001_SN51 [1]
   RUNG wire#powerrail
      "n0091-zp001-el001-k30001_SN51_1"(IN_1 := "EMERGENCY PUSH BUTTON PRESSED =SE01+NA0078-S1", IN_2 := "EMERGENCY PUSH BUTTON PRESSED =SE01+NA0079-S1", IN_3 := "EMERGENCY PUSH BUTTON PRESSED =SE01+NA0080-S1", IN_4 := "EMERGENCY PUSH BUTTON PRESSED =SE01+NA0081-S1", ON_Tristate := "06_Settings".Tristate, ON_Lamp :=, Reset :=, REAC_DELAY :=, Bypass_ET200 := "00_Commissioning"."n0091-zp001-el001-k30001_SN51", OUT_1 => "01_PushButton"."SE01+NA0078-S1_PB", OUT_2 => "01_PushButton"."SE01+NA0079-S1_PB", OUT_3 => "01_PushButton"."SE01+NA0080-S1_PB", OUT_4 => "01_PushButton"."SE01+NA0081-S1_PB", Diag_1 =>, Diag_2 =>, Diag_3 =>, Diag_4 =>, Lamp_1 =>, Lamp_2 =>, Lamp_3 =>, Lamp_4 =>)
   END_RUNG
   // the same network as SCL:
   "n0091-zp001-el001-k30001_SN51_1"(IN_1 := "EMERGENCY PUSH BUTTON PRESSED =SE01+NA0078-S1",   // "00_Push-Button_Input"
                           IN_2 := "EMERGENCY PUSH BUTTON PRESSED =SE01+NA0079-S1",
                           IN_3 := "EMERGENCY PUSH BUTTON PRESSED =SE01+NA0080-S1",
                           IN_4 := "EMERGENCY PUSH BUTTON PRESSED =SE01+NA0081-S1",
                           ON_Tristate := "06_Settings".Tristate,
                           Bypass_ET200 := "00_Commissioning"."n0091-zp001-el001-k30001_SN51",
                           OUT_1 => "01_PushButton"."SE01+NA0078-S1_PB",
                           OUT_2 => "01_PushButton"."SE01+NA0079-S1_PB",
                           OUT_3 => "01_PushButton"."SE01+NA0080-S1_PB",
                           OUT_4 => "01_PushButton"."SE01+NA0081-S1_PB");
END_REGION

REGION Network 145: 51.091 | n0091-zp001-el001-k30001_SN51 [2]
   RUNG wire#powerrail
      "n0091-zp001-el001-k30001_SN51_2"(IN_1 := "EMERGENCY PUSH BUTTON PRESSED =SE01+NA0082-S1", IN_2 := "EMERGENCY PUSH BUTTON PRESSED =SG06+ZP001.EL001-S31001", IN_3 := "EMERGENCY PUSH BUTTON PRESSED =SE01+NA0015-S1", IN_4 := "EMERGENCY PUSH BUTTON PRESSED =SE01+NA0016-S1", ON_Tristate := "06_Settings".Tristate, ON_Lamp :=, Reset :=, REAC_DELAY :=, Bypass_ET200 := "00_Commissioning"."n0091-zp001-el001-k30001_SN51", OUT_1 => "01_PushButton"."SE01+NA0082-S1_PB", OUT_2 => "01_PushButton"."SG06+ZP001.EL001-S31001_PB", OUT_3 => "01_PushButton"."SE01+NA0015-S1_PB", OUT_4 => "01_PushButton"."SE01+NA0016-S1_PB", Diag_1 =>, Diag_2 =>, Diag_3 =>, Diag_4 =>, Lamp_1 =>, Lamp_2 =>, Lamp_3 =>, Lamp_4 =>)
   END_RUNG
   // the same network as SCL:
   "n0091-zp001-el001-k30001_SN51_2"(IN_1 := "EMERGENCY PUSH BUTTON PRESSED =SE01+NA0082-S1",   // "00_Push-Button_Input"
                           IN_2 := "EMERGENCY PUSH BUTTON PRESSED =SG06+ZP001.EL001-S31001",
                           IN_3 := "EMERGENCY PUSH BUTTON PRESSED =SE01+NA0015-S1",
                           IN_4 := "EMERGENCY PUSH BUTTON PRESSED =SE01+NA0016-S1",
                           ON_Tristate := "06_Settings".Tristate,
                           Bypass_ET200 := "00_Commissioning"."n0091-zp001-el001-k30001_SN51",
                           OUT_1 => "01_PushButton"."SE01+NA0082-S1_PB",
                           OUT_2 => "01_PushButton"."SG06+ZP001.EL001-S31001_PB",
                           OUT_3 => "01_PushButton"."SE01+NA0015-S1_PB",
                           OUT_4 => "01_PushButton"."SE01+NA0016-S1_PB");
END_REGION

REGION Network 146: 51.091 | n0091-zp001-el001-k30001_SN51 [3]
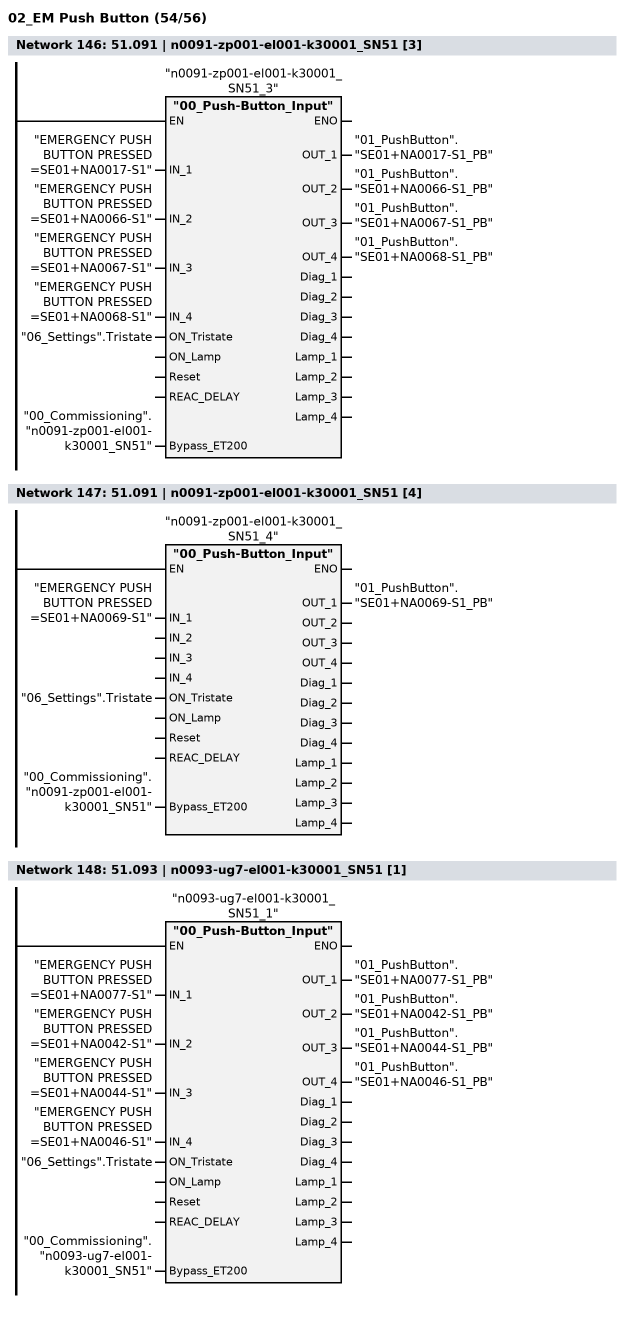
   RUNG wire#powerrail
      "n0091-zp001-el001-k30001_SN51_3"(IN_1 := "EMERGENCY PUSH BUTTON PRESSED =SE01+NA0017-S1", IN_2 := "EMERGENCY PUSH BUTTON PRESSED =SE01+NA0066-S1", IN_3 := "EMERGENCY PUSH BUTTON PRESSED =SE01+NA0067-S1", IN_4 := "EMERGENCY PUSH BUTTON PRESSED =SE01+NA0068-S1", ON_Tristate := "06_Settings".Tristate, ON_Lamp :=, Reset :=, REAC_DELAY :=, Bypass_ET200 := "00_Commissioning"."n0091-zp001-el001-k30001_SN51", OUT_1 => "01_PushButton"."SE01+NA0017-S1_PB", OUT_2 => "01_PushButton"."SE01+NA0066-S1_PB", OUT_3 => "01_PushButton"."SE01+NA0067-S1_PB", OUT_4 => "01_PushButton"."SE01+NA0068-S1_PB", Diag_1 =>, Diag_2 =>, Diag_3 =>, Diag_4 =>, Lamp_1 =>, Lamp_2 =>, Lamp_3 =>, Lamp_4 =>)
   END_RUNG
   // the same network as SCL:
   "n0091-zp001-el001-k30001_SN51_3"(IN_1 := "EMERGENCY PUSH BUTTON PRESSED =SE01+NA0017-S1",   // "00_Push-Button_Input"
                           IN_2 := "EMERGENCY PUSH BUTTON PRESSED =SE01+NA0066-S1",
                           IN_3 := "EMERGENCY PUSH BUTTON PRESSED =SE01+NA0067-S1",
                           IN_4 := "EMERGENCY PUSH BUTTON PRESSED =SE01+NA0068-S1",
                           ON_Tristate := "06_Settings".Tristate,
                           Bypass_ET200 := "00_Commissioning"."n0091-zp001-el001-k30001_SN51",
                           OUT_1 => "01_PushButton"."SE01+NA0017-S1_PB",
                           OUT_2 => "01_PushButton"."SE01+NA0066-S1_PB",
                           OUT_3 => "01_PushButton"."SE01+NA0067-S1_PB",
                           OUT_4 => "01_PushButton"."SE01+NA0068-S1_PB");
END_REGION

REGION Network 147: 51.091 | n0091-zp001-el001-k30001_SN51 [4]
   RUNG wire#powerrail
      "n0091-zp001-el001-k30001_SN51_4"(IN_1 := "EMERGENCY PUSH BUTTON PRESSED =SE01+NA0069-S1", IN_2 :=, IN_3 :=, IN_4 :=, ON_Tristate := "06_Settings".Tristate, ON_Lamp :=, Reset :=, REAC_DELAY :=, Bypass_ET200 := "00_Commissioning"."n0091-zp001-el001-k30001_SN51", OUT_1 => "01_PushButton"."SE01+NA0069-S1_PB", OUT_2 =>, OUT_3 =>, OUT_4 =>, Diag_1 =>, Diag_2 =>, Diag_3 =>, Diag_4 =>, Lamp_1 =>, Lamp_2 =>, Lamp_3 =>, Lamp_4 =>)
   END_RUNG
   // the same network as SCL:
   "n0091-zp001-el001-k30001_SN51_4"(IN_1 := "EMERGENCY PUSH BUTTON PRESSED =SE01+NA0069-S1",   // "00_Push-Button_Input"
                           ON_Tristate := "06_Settings".Tristate,
                           Bypass_ET200 := "00_Commissioning"."n0091-zp001-el001-k30001_SN51",
                           OUT_1 => "01_PushButton"."SE01+NA0069-S1_PB");
END_REGION

REGION Network 148: 51.093 | n0093-ug7-el001-k30001_SN51 [1]
   RUNG wire#powerrail
      "n0093-ug7-el001-k30001_SN51_1"(IN_1 := "EMERGENCY PUSH BUTTON PRESSED =SE01+NA0077-S1", IN_2 := "EMERGENCY PUSH BUTTON PRESSED =SE01+NA0042-S1", IN_3 := "EMERGENCY PUSH BUTTON PRESSED =SE01+NA0044-S1", IN_4 := "EMERGENCY PUSH BUTTON PRESSED =SE01+NA0046-S1", ON_Tristate := "06_Settings".Tristate, ON_Lamp :=, Reset :=, REAC_DELAY :=, Bypass_ET200 := "00_Commissioning"."n0093-ug7-el001-k30001_SN51", OUT_1 => "01_PushButton"."SE01+NA0077-S1_PB", OUT_2 => "01_PushButton"."SE01+NA0042-S1_PB", OUT_3 => "01_PushButton"."SE01+NA0044-S1_PB", OUT_4 => "01_PushButton"."SE01+NA0046-S1_PB", Diag_1 =>, Diag_2 =>, Diag_3 =>, Diag_4 =>, Lamp_1 =>, Lamp_2 =>, Lamp_3 =>, Lamp_4 =>)
   END_RUNG
   // the same network as SCL:
   "n0093-ug7-el001-k30001_SN51_1"(IN_1 := "EMERGENCY PUSH BUTTON PRESSED =SE01+NA0077-S1",   // "00_Push-Button_Input"
                           IN_2 := "EMERGENCY PUSH BUTTON PRESSED =SE01+NA0042-S1",
                           IN_3 := "EMERGENCY PUSH BUTTON PRESSED =SE01+NA0044-S1",
                           IN_4 := "EMERGENCY PUSH BUTTON PRESSED =SE01+NA0046-S1",
                           ON_Tristate := "06_Settings".Tristate,
                           Bypass_ET200 := "00_Commissioning"."n0093-ug7-el001-k30001_SN51",
                           OUT_1 => "01_PushButton"."SE01+NA0077-S1_PB",
                           OUT_2 => "01_PushButton"."SE01+NA0042-S1_PB",
                           OUT_3 => "01_PushButton"."SE01+NA0044-S1_PB",
                           OUT_4 => "01_PushButton"."SE01+NA0046-S1_PB");
END_REGION

REGION Network 149: 51.093 | n0093-ug7-el001-k30001_SN51 [2]
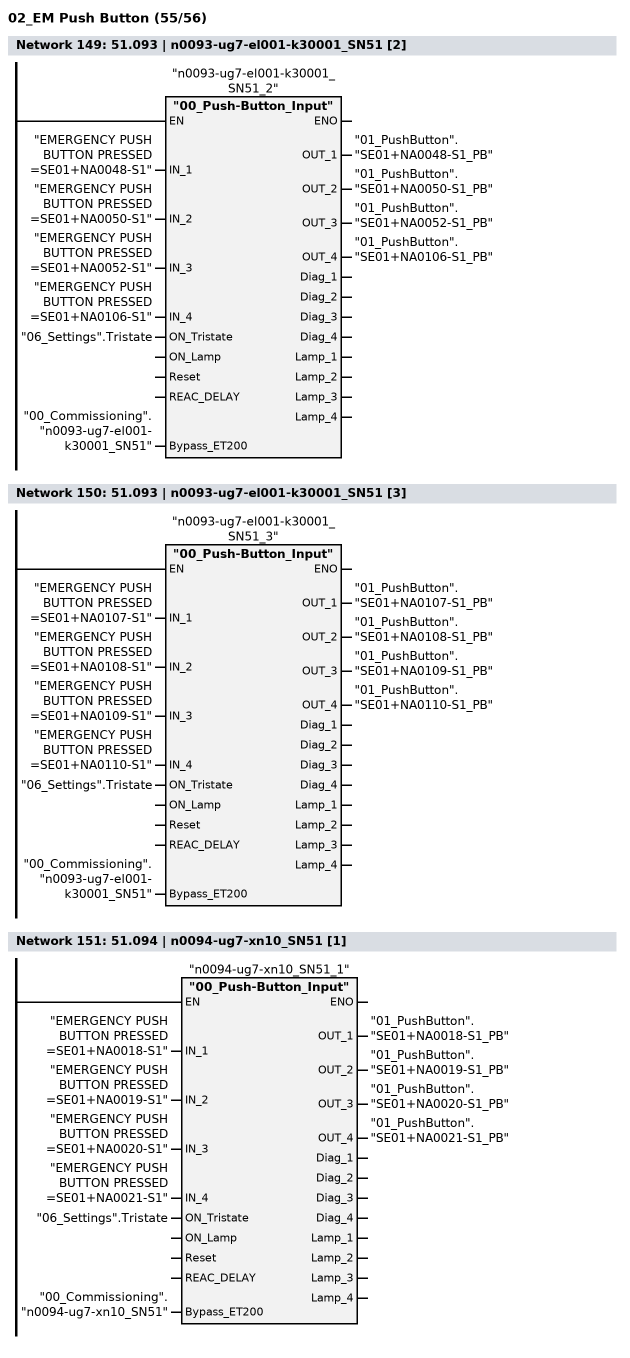
   RUNG wire#powerrail
      "n0093-ug7-el001-k30001_SN51_2"(IN_1 := "EMERGENCY PUSH BUTTON PRESSED =SE01+NA0048-S1", IN_2 := "EMERGENCY PUSH BUTTON PRESSED =SE01+NA0050-S1", IN_3 := "EMERGENCY PUSH BUTTON PRESSED =SE01+NA0052-S1", IN_4 := "EMERGENCY PUSH BUTTON PRESSED =SE01+NA0106-S1", ON_Tristate := "06_Settings".Tristate, ON_Lamp :=, Reset :=, REAC_DELAY :=, Bypass_ET200 := "00_Commissioning"."n0093-ug7-el001-k30001_SN51", OUT_1 => "01_PushButton"."SE01+NA0048-S1_PB", OUT_2 => "01_PushButton"."SE01+NA0050-S1_PB", OUT_3 => "01_PushButton"."SE01+NA0052-S1_PB", OUT_4 => "01_PushButton"."SE01+NA0106-S1_PB", Diag_1 =>, Diag_2 =>, Diag_3 =>, Diag_4 =>, Lamp_1 =>, Lamp_2 =>, Lamp_3 =>, Lamp_4 =>)
   END_RUNG
   // the same network as SCL:
   "n0093-ug7-el001-k30001_SN51_2"(IN_1 := "EMERGENCY PUSH BUTTON PRESSED =SE01+NA0048-S1",   // "00_Push-Button_Input"
                           IN_2 := "EMERGENCY PUSH BUTTON PRESSED =SE01+NA0050-S1",
                           IN_3 := "EMERGENCY PUSH BUTTON PRESSED =SE01+NA0052-S1",
                           IN_4 := "EMERGENCY PUSH BUTTON PRESSED =SE01+NA0106-S1",
                           ON_Tristate := "06_Settings".Tristate,
                           Bypass_ET200 := "00_Commissioning"."n0093-ug7-el001-k30001_SN51",
                           OUT_1 => "01_PushButton"."SE01+NA0048-S1_PB",
                           OUT_2 => "01_PushButton"."SE01+NA0050-S1_PB",
                           OUT_3 => "01_PushButton"."SE01+NA0052-S1_PB",
                           OUT_4 => "01_PushButton"."SE01+NA0106-S1_PB");
END_REGION

REGION Network 150: 51.093 | n0093-ug7-el001-k30001_SN51 [3]
   RUNG wire#powerrail
      "n0093-ug7-el001-k30001_SN51_3"(IN_1 := "EMERGENCY PUSH BUTTON PRESSED =SE01+NA0107-S1", IN_2 := "EMERGENCY PUSH BUTTON PRESSED =SE01+NA0108-S1", IN_3 := "EMERGENCY PUSH BUTTON PRESSED =SE01+NA0109-S1", IN_4 := "EMERGENCY PUSH BUTTON PRESSED =SE01+NA0110-S1", ON_Tristate := "06_Settings".Tristate, ON_Lamp :=, Reset :=, REAC_DELAY :=, Bypass_ET200 := "00_Commissioning"."n0093-ug7-el001-k30001_SN51", OUT_1 => "01_PushButton"."SE01+NA0107-S1_PB", OUT_2 => "01_PushButton"."SE01+NA0108-S1_PB", OUT_3 => "01_PushButton"."SE01+NA0109-S1_PB", OUT_4 => "01_PushButton"."SE01+NA0110-S1_PB", Diag_1 =>, Diag_2 =>, Diag_3 =>, Diag_4 =>, Lamp_1 =>, Lamp_2 =>, Lamp_3 =>, Lamp_4 =>)
   END_RUNG
   // the same network as SCL:
   "n0093-ug7-el001-k30001_SN51_3"(IN_1 := "EMERGENCY PUSH BUTTON PRESSED =SE01+NA0107-S1",   // "00_Push-Button_Input"
                           IN_2 := "EMERGENCY PUSH BUTTON PRESSED =SE01+NA0108-S1",
                           IN_3 := "EMERGENCY PUSH BUTTON PRESSED =SE01+NA0109-S1",
                           IN_4 := "EMERGENCY PUSH BUTTON PRESSED =SE01+NA0110-S1",
                           ON_Tristate := "06_Settings".Tristate,
                           Bypass_ET200 := "00_Commissioning"."n0093-ug7-el001-k30001_SN51",
                           OUT_1 => "01_PushButton"."SE01+NA0107-S1_PB",
                           OUT_2 => "01_PushButton"."SE01+NA0108-S1_PB",
                           OUT_3 => "01_PushButton"."SE01+NA0109-S1_PB",
                           OUT_4 => "01_PushButton"."SE01+NA0110-S1_PB");
END_REGION

REGION Network 151: 51.094 | n0094-ug7-xn10_SN51 [1]
   RUNG wire#powerrail
      "n0094-ug7-xn10_SN51_1"(IN_1 := "EMERGENCY PUSH BUTTON PRESSED =SE01+NA0018-S1", IN_2 := "EMERGENCY PUSH BUTTON PRESSED =SE01+NA0019-S1", IN_3 := "EMERGENCY PUSH BUTTON PRESSED =SE01+NA0020-S1", IN_4 := "EMERGENCY PUSH BUTTON PRESSED =SE01+NA0021-S1", ON_Tristate := "06_Settings".Tristate, ON_Lamp :=, Reset :=, REAC_DELAY :=, Bypass_ET200 := "00_Commissioning"."n0094-ug7-xn10_SN51", OUT_1 => "01_PushButton"."SE01+NA0018-S1_PB", OUT_2 => "01_PushButton"."SE01+NA0019-S1_PB", OUT_3 => "01_PushButton"."SE01+NA0020-S1_PB", OUT_4 => "01_PushButton"."SE01+NA0021-S1_PB", Diag_1 =>, Diag_2 =>, Diag_3 =>, Diag_4 =>, Lamp_1 =>, Lamp_2 =>, Lamp_3 =>, Lamp_4 =>)
   END_RUNG
   // the same network as SCL:
   "n0094-ug7-xn10_SN51_1"(IN_1 := "EMERGENCY PUSH BUTTON PRESSED =SE01+NA0018-S1",   // "00_Push-Button_Input"
                           IN_2 := "EMERGENCY PUSH BUTTON PRESSED =SE01+NA0019-S1",
                           IN_3 := "EMERGENCY PUSH BUTTON PRESSED =SE01+NA0020-S1",
                           IN_4 := "EMERGENCY PUSH BUTTON PRESSED =SE01+NA0021-S1",
                           ON_Tristate := "06_Settings".Tristate,
                           Bypass_ET200 := "00_Commissioning"."n0094-ug7-xn10_SN51",
                           OUT_1 => "01_PushButton"."SE01+NA0018-S1_PB",
                           OUT_2 => "01_PushButton"."SE01+NA0019-S1_PB",
                           OUT_3 => "01_PushButton"."SE01+NA0020-S1_PB",
                           OUT_4 => "01_PushButton"."SE01+NA0021-S1_PB");
END_REGION

REGION Network 152: 51.094 | n0094-ug7-xn10_SN51 [2]
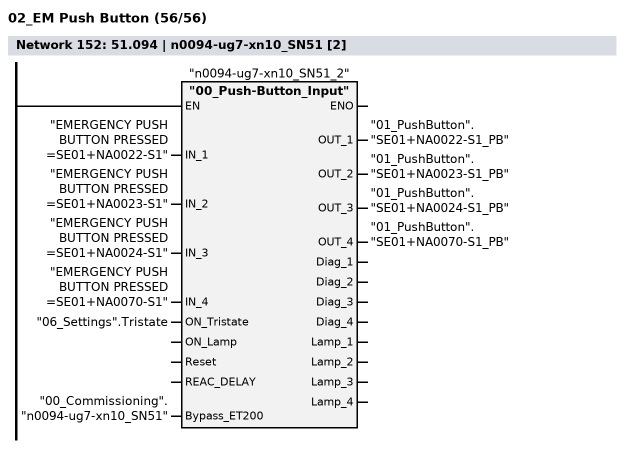
   RUNG wire#powerrail
      "n0094-ug7-xn10_SN51_2"(IN_1 := "EMERGENCY PUSH BUTTON PRESSED =SE01+NA0022-S1", IN_2 := "EMERGENCY PUSH BUTTON PRESSED =SE01+NA0023-S1", IN_3 := "EMERGENCY PUSH BUTTON PRESSED =SE01+NA0024-S1", IN_4 := "EMERGENCY PUSH BUTTON PRESSED =SE01+NA0070-S1", ON_Tristate := "06_Settings".Tristate, ON_Lamp :=, Reset :=, REAC_DELAY :=, Bypass_ET200 := "00_Commissioning"."n0094-ug7-xn10_SN51", OUT_1 => "01_PushButton"."SE01+NA0022-S1_PB", OUT_2 => "01_PushButton"."SE01+NA0023-S1_PB", OUT_3 => "01_PushButton"."SE01+NA0024-S1_PB", OUT_4 => "01_PushButton"."SE01+NA0070-S1_PB", Diag_1 =>, Diag_2 =>, Diag_3 =>, Diag_4 =>, Lamp_1 =>, Lamp_2 =>, Lamp_3 =>, Lamp_4 =>)
   END_RUNG
   // the same network as SCL:
   "n0094-ug7-xn10_SN51_2"(IN_1 := "EMERGENCY PUSH BUTTON PRESSED =SE01+NA0022-S1",   // "00_Push-Button_Input"
                           IN_2 := "EMERGENCY PUSH BUTTON PRESSED =SE01+NA0023-S1",
                           IN_3 := "EMERGENCY PUSH BUTTON PRESSED =SE01+NA0024-S1",
                           IN_4 := "EMERGENCY PUSH BUTTON PRESSED =SE01+NA0070-S1",
                           ON_Tristate := "06_Settings".Tristate,
                           Bypass_ET200 := "00_Commissioning"."n0094-ug7-xn10_SN51",
                           OUT_1 => "01_PushButton"."SE01+NA0022-S1_PB",
                           OUT_2 => "01_PushButton"."SE01+NA0023-S1_PB",
                           OUT_3 => "01_PushButton"."SE01+NA0024-S1_PB",
                           OUT_4 => "01_PushButton"."SE01+NA0070-S1_PB");
END_REGION
END_FUNCTION

FUNCTION "03_Zone Cumulative" : Void   // FC4, F_FBD
{ S7_Optimized_Access := 'TRUE' }
VERSION : 0.1
BEGIN

REGION Network 1: S1 PB | ^SORTER UPPER COY =SC01
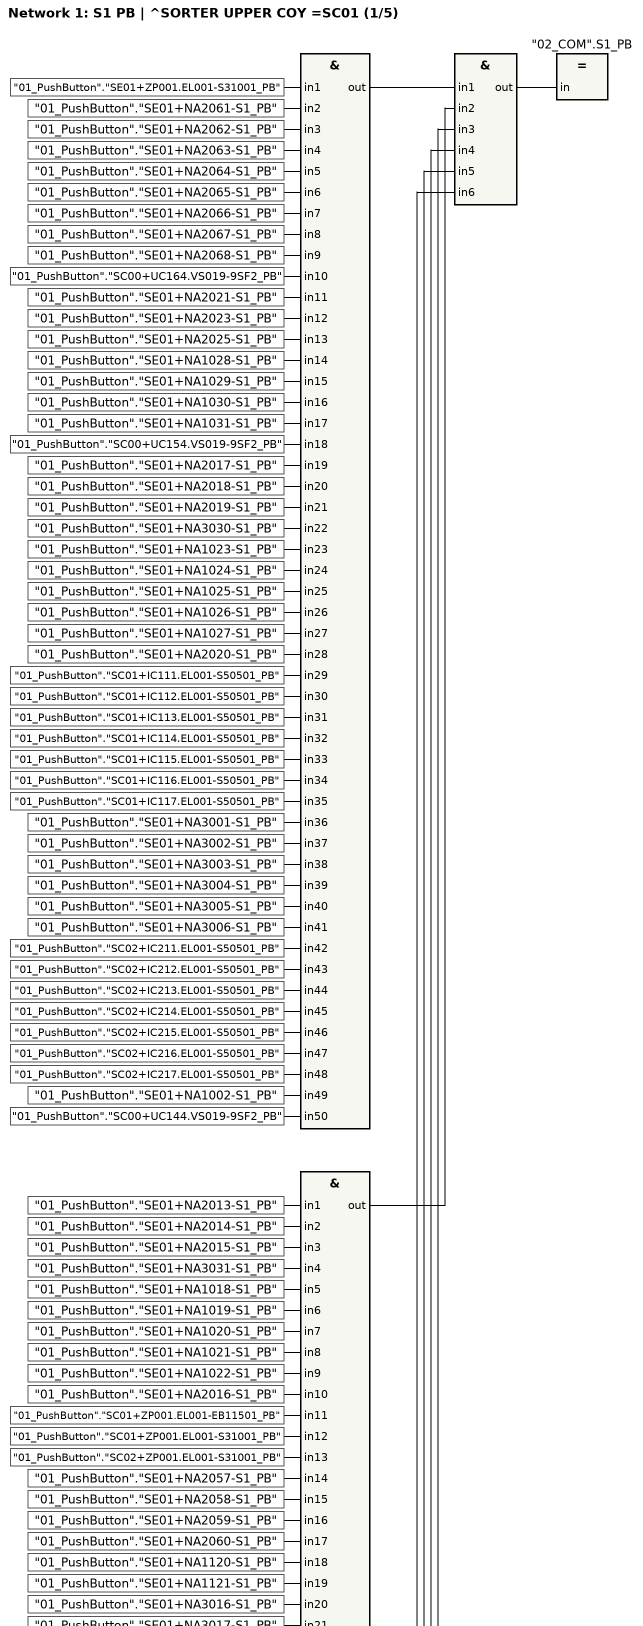
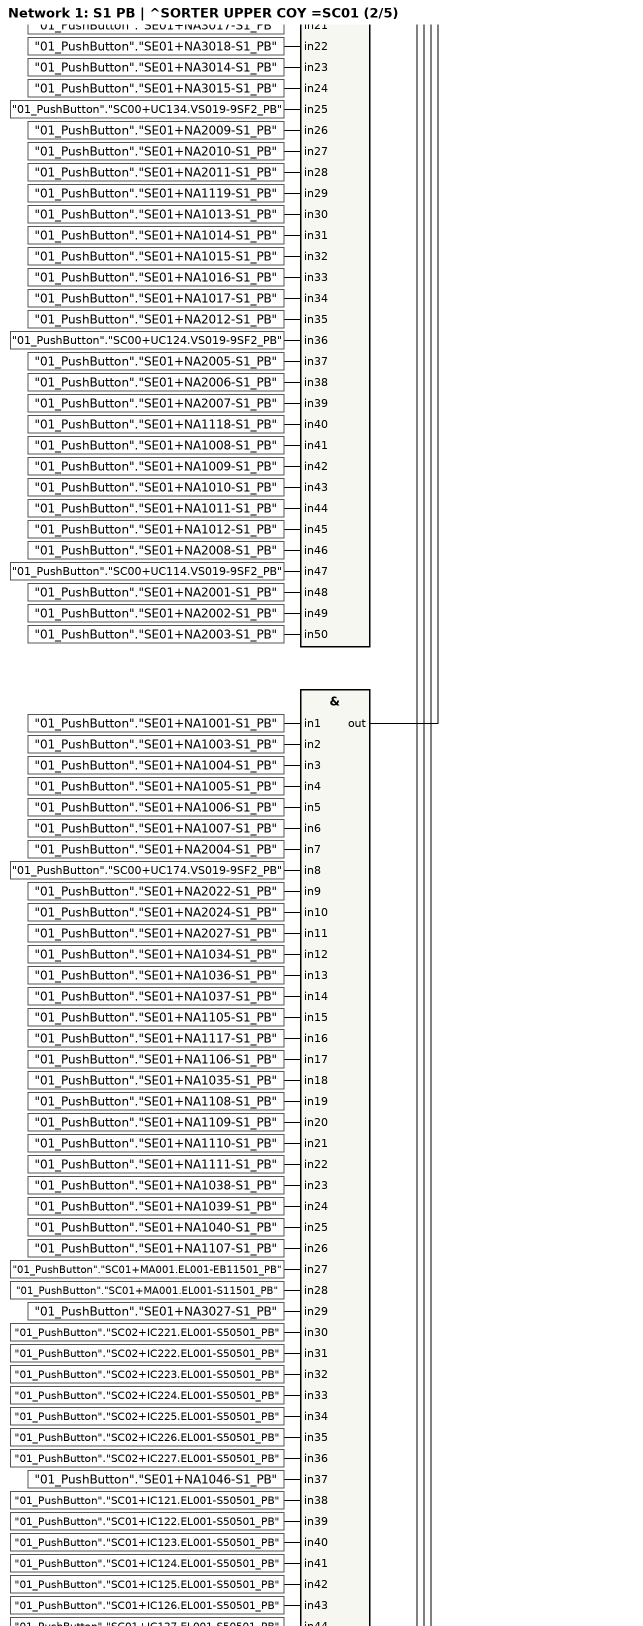
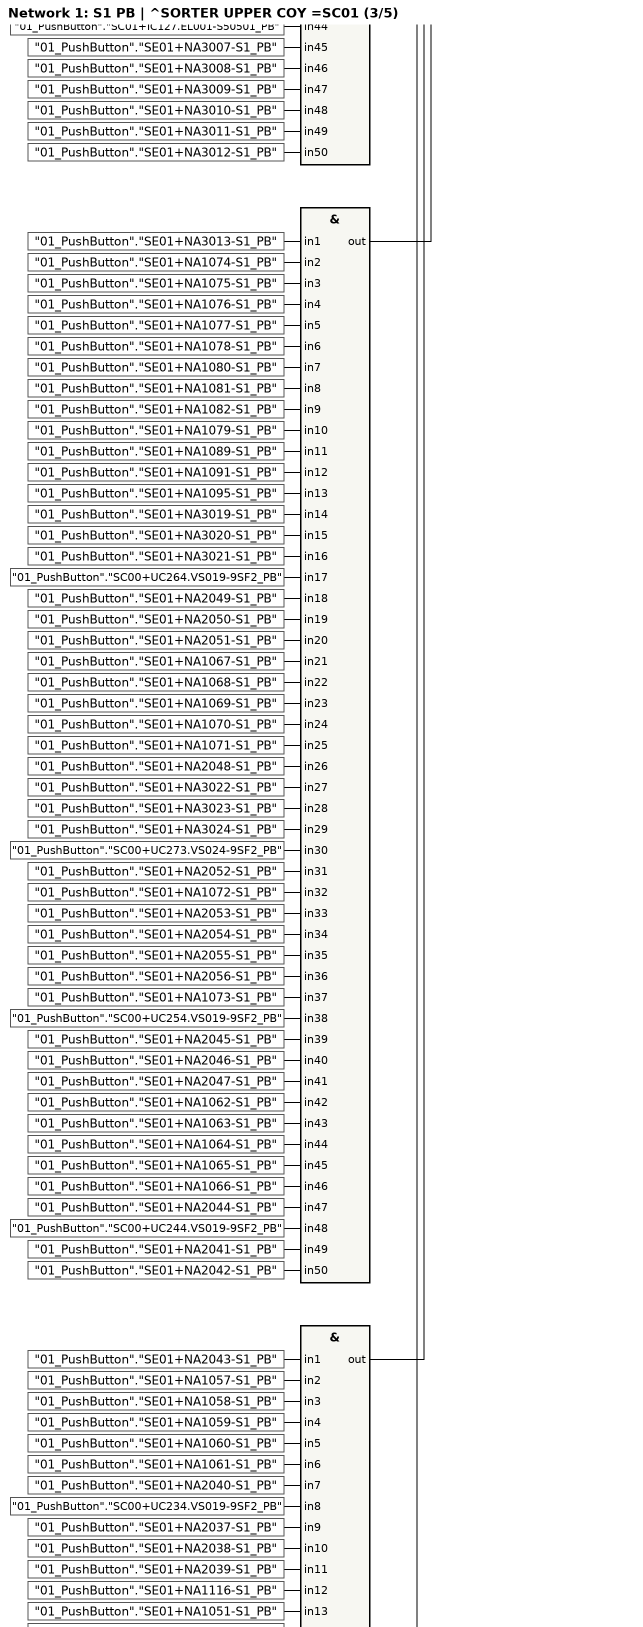
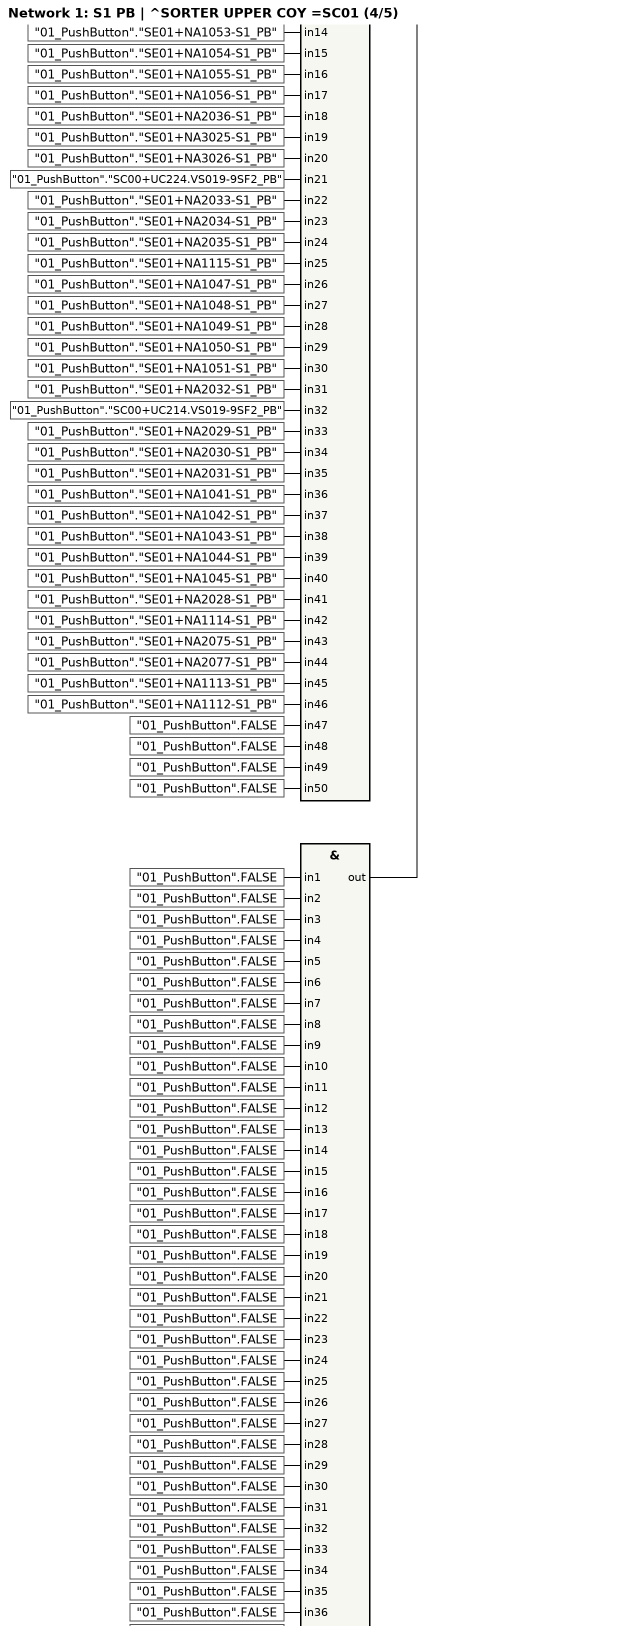
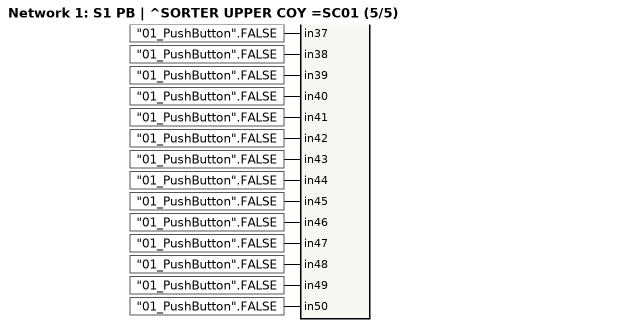
   "02_COM".S1_PB := "01_PushButton"."SE01+ZP001.EL001-S31001_PB" AND "01_PushButton"."SE01+NA2061-S1_PB" AND "01_PushButton"."SE01+NA2062-S1_PB" AND "01_PushButton"."SE01+NA2063-S1_PB" AND "01_PushButton"."SE01+NA2064-S1_PB" AND "01_PushButton"."SE01+NA2065-S1_PB" AND "01_PushButton"."SE01+NA2066-S1_PB" AND "01_PushButton"."SE01+NA2067-S1_PB" AND "01_PushButton"."SE01+NA2068-S1_PB" AND "01_PushButton"."SC00+UC164.VS019-9SF2_PB" AND "01_PushButton"."SE01+NA2021-S1_PB" AND "01_PushButton"."SE01+NA2023-S1_PB" AND "01_PushButton"."SE01+NA2025-S1_PB" AND "01_PushButton"."SE01+NA1028-S1_PB" AND "01_PushButton"."SE01+NA1029-S1_PB" AND "01_PushButton"."SE01+NA1030-S1_PB" AND "01_PushButton"."SE01+NA1031-S1_PB" AND "01_PushButton"."SC00+UC154.VS019-9SF2_PB" AND "01_PushButton"."SE01+NA2017-S1_PB" AND "01_PushButton"."SE01+NA2018-S1_PB" AND "01_PushButton"."SE01+NA2019-S1_PB" AND "01_PushButton"."SE01+NA3030-S1_PB" AND "01_PushButton"."SE01+NA1023-S1_PB" AND "01_PushButton"."SE01+NA1024-S1_PB" AND "01_PushButton"."SE01+NA1025-S1_PB" AND "01_PushButton"."SE01+NA1026-S1_PB" AND "01_PushButton"."SE01+NA1027-S1_PB" AND "01_PushButton"."SE01+NA2020-S1_PB" AND "01_PushButton"."SC01+IC111.EL001-S50501_PB" AND "01_PushButton"."SC01+IC112.EL001-S50501_PB" AND "01_PushButton"."SC01+IC113.EL001-S50501_PB" AND "01_PushButton"."SC01+IC114.EL001-S50501_PB" AND "01_PushButton"."SC01+IC115.EL001-S50501_PB" AND "01_PushButton"."SC01+IC116.EL001-S50501_PB" AND "01_PushButton"."SC01+IC117.EL001-S50501_PB" AND "01_PushButton"."SE01+NA3001-S1_PB" AND "01_PushButton"."SE01+NA3002-S1_PB" AND "01_PushButton"."SE01+NA3003-S1_PB" AND "01_PushButton"."SE01+NA3004-S1_PB" AND "01_PushButton"."SE01+NA3005-S1_PB" AND "01_PushButton"."SE01+NA3006-S1_PB" AND "01_PushButton"."SC02+IC211.EL001-S50501_PB" AND "01_PushButton"."SC02+IC212.EL001-S50501_PB" AND "01_PushButton"."SC02+IC213.EL001-S50501_PB" AND "01_PushButton"."SC02+IC214.EL001-S50501_PB" AND "01_PushButton"."SC02+IC215.EL001-S50501_PB" AND "01_PushButton"."SC02+IC216.EL001-S50501_PB" AND "01_PushButton"."SC02+IC217.EL001-S50501_PB" AND "01_PushButton"."SE01+NA1002-S1_PB" AND "01_PushButton"."SC00+UC144.VS019-9SF2_PB" AND "01_PushButton"."SE01+NA2013-S1_PB" AND "01_PushButton"."SE01+NA2014-S1_PB" AND "01_PushButton"."SE01+NA2015-S1_PB" AND "01_PushButton"."SE01+NA3031-S1_PB" AND "01_PushButton"."SE01+NA1018-S1_PB" AND "01_PushButton"."SE01+NA1019-S1_PB" AND "01_PushButton"."SE01+NA1020-S1_PB" AND "01_PushButton"."SE01+NA1021-S1_PB" AND "01_PushButton"."SE01+NA1022-S1_PB" AND "01_PushButton"."SE01+NA2016-S1_PB" AND "01_PushButton"."SC01+ZP001.EL001-EB11501_PB" AND "01_PushButton"."SC01+ZP001.EL001-S31001_PB" AND "01_PushButton"."SC02+ZP001.EL001-S31001_PB" AND "01_PushButton"."SE01+NA2057-S1_PB" AND "01_PushButton"."SE01+NA2058-S1_PB" AND "01_PushButton"."SE01+NA2059-S1_PB" AND "01_PushButton"."SE01+NA2060-S1_PB" AND "01_PushButton"."SE01+NA1120-S1_PB" AND "01_PushButton"."SE01+NA1121-S1_PB" AND "01_PushButton"."SE01+NA3016-S1_PB" AND "01_PushButton"."SE01+NA3017-S1_PB" AND "01_PushButton"."SE01+NA3018-S1_PB" AND "01_PushButton"."SE01+NA3014-S1_PB" AND "01_PushButton"."SE01+NA3015-S1_PB" AND "01_PushButton"."SC00+UC134.VS019-9SF2_PB" AND "01_PushButton"."SE01+NA2009-S1_PB" AND "01_PushButton"."SE01+NA2010-S1_PB" AND "01_PushButton"."SE01+NA2011-S1_PB" AND "01_PushButton"."SE01+NA1119-S1_PB" AND "01_PushButton"."SE01+NA1013-S1_PB" AND "01_PushButton"."SE01+NA1014-S1_PB" AND "01_PushButton"."SE01+NA1015-S1_PB" AND "01_PushButton"."SE01+NA1016-S1_PB" AND "01_PushButton"."SE01+NA1017-S1_PB" AND "01_PushButton"."SE01+NA2012-S1_PB" AND "01_PushButton"."SC00+UC124.VS019-9SF2_PB" AND "01_PushButton"."SE01+NA2005-S1_PB" AND "01_PushButton"."SE01+NA2006-S1_PB" AND "01_PushButton"."SE01+NA2007-S1_PB" AND "01_PushButton"."SE01+NA1118-S1_PB" AND "01_PushButton"."SE01+NA1008-S1_PB" AND "01_PushButton"."SE01+NA1009-S1_PB" AND "01_PushButton"."SE01+NA1010-S1_PB" AND "01_PushButton"."SE01+NA1011-S1_PB" AND "01_PushButton"."SE01+NA1012-S1_PB" AND "01_PushButton"."SE01+NA2008-S1_PB" AND "01_PushButton"."SC00+UC114.VS019-9SF2_PB" AND "01_PushButton"."SE01+NA2001-S1_PB" AND "01_PushButton"."SE01+NA2002-S1_PB" AND "01_PushButton"."SE01+NA2003-S1_PB" AND "01_PushButton"."SE01+NA1001-S1_PB" AND "01_PushButton"."SE01+NA1003-S1_PB" AND "01_PushButton"."SE01+NA1004-S1_PB" AND "01_PushButton"."SE01+NA1005-S1_PB" AND "01_PushButton"."SE01+NA1006-S1_PB" AND "01_PushButton"."SE01+NA1007-S1_PB" AND "01_PushButton"."SE01+NA2004-S1_PB" AND "01_PushButton"."SC00+UC174.VS019-9SF2_PB" AND "01_PushButton"."SE01+NA2022-S1_PB" AND "01_PushButton"."SE01+NA2024-S1_PB" AND "01_PushButton"."SE01+NA2027-S1_PB" AND "01_PushButton"."SE01+NA1034-S1_PB" AND "01_PushButton"."SE01+NA1036-S1_PB" AND "01_PushButton"."SE01+NA1037-S1_PB" AND "01_PushButton"."SE01+NA1105-S1_PB" AND "01_PushButton"."SE01+NA1117-S1_PB" AND "01_PushButton"."SE01+NA1106-S1_PB" AND "01_PushButton"."SE01+NA1035-S1_PB" AND "01_PushButton"."SE01+NA1108-S1_PB" AND "01_PushButton"."SE01+NA1109-S1_PB" AND "01_PushButton"."SE01+NA1110-S1_PB" AND "01_PushButton"."SE01+NA1111-S1_PB" AND "01_PushButton"."SE01+NA1038-S1_PB" AND "01_PushButton"."SE01+NA1039-S1_PB" AND "01_PushButton"."SE01+NA1040-S1_PB" AND "01_PushButton"."SE01+NA1107-S1_PB" AND "01_PushButton"."SC01+MA001.EL001-EB11501_PB" AND "01_PushButton"."SC01+MA001.EL001-S11501_PB" AND "01_PushButton"."SE01+NA3027-S1_PB" AND "01_PushButton"."SC02+IC221.EL001-S50501_PB" AND "01_PushButton"."SC02+IC222.EL001-S50501_PB" AND "01_PushButton"."SC02+IC223.EL001-S50501_PB" AND "01_PushButton"."SC02+IC224.EL001-S50501_PB" AND "01_PushButton"."SC02+IC225.EL001-S50501_PB" AND "01_PushButton"."SC02+IC226.EL001-S50501_PB" AND "01_PushButton"."SC02+IC227.EL001-S50501_PB" AND "01_PushButton"."SE01+NA1046-S1_PB" AND "01_PushButton"."SC01+IC121.EL001-S50501_PB" AND "01_PushButton"."SC01+IC122.EL001-S50501_PB" AND "01_PushButton"."SC01+IC123.EL001-S50501_PB" AND "01_PushButton"."SC01+IC124.EL001-S50501_PB" AND "01_PushButton"."SC01+IC125.EL001-S50501_PB" AND "01_PushButton"."SC01+IC126.EL001-S50501_PB" AND "01_PushButton"."SC01+IC127.EL001-S50501_PB" AND "01_PushButton"."SE01+NA3007-S1_PB" AND "01_PushButton"."SE01+NA3008-S1_PB" AND "01_PushButton"."SE01+NA3009-S1_PB" AND "01_PushButton"."SE01+NA3010-S1_PB" AND "01_PushButton"."SE01+NA3011-S1_PB" AND "01_PushButton"."SE01+NA3012-S1_PB" AND "01_PushButton"."SE01+NA3013-S1_PB" AND "01_PushButton"."SE01+NA1074-S1_PB" AND "01_PushButton"."SE01+NA1075-S1_PB" AND "01_PushButton"."SE01+NA1076-S1_PB" AND "01_PushButton"."SE01+NA1077-S1_PB" AND "01_PushButton"."SE01+NA1078-S1_PB" AND "01_PushButton"."SE01+NA1080-S1_PB" AND "01_PushButton"."SE01+NA1081-S1_PB" AND "01_PushButton"."SE01+NA1082-S1_PB" AND "01_PushButton"."SE01+NA1079-S1_PB" AND "01_PushButton"."SE01+NA1089-S1_PB" AND "01_PushButton"."SE01+NA1091-S1_PB" AND "01_PushButton"."SE01+NA1095-S1_PB" AND "01_PushButton"."SE01+NA3019-S1_PB" AND "01_PushButton"."SE01+NA3020-S1_PB" AND "01_PushButton"."SE01+NA3021-S1_PB" AND "01_PushButton"."SC00+UC264.VS019-9SF2_PB" AND "01_PushButton"."SE01+NA2049-S1_PB" AND "01_PushButton"."SE01+NA2050-S1_PB" AND "01_PushButton"."SE01+NA2051-S1_PB" AND "01_PushButton"."SE01+NA1067-S1_PB" AND "01_PushButton"."SE01+NA1068-S1_PB" AND "01_PushButton"."SE01+NA1069-S1_PB" AND "01_PushButton"."SE01+NA1070-S1_PB" AND "01_PushButton"."SE01+NA1071-S1_PB" AND "01_PushButton"."SE01+NA2048-S1_PB" AND "01_PushButton"."SE01+NA3022-S1_PB" AND "01_PushButton"."SE01+NA3023-S1_PB" AND "01_PushButton"."SE01+NA3024-S1_PB" AND "01_PushButton"."SC00+UC273.VS024-9SF2_PB" AND "01_PushButton"."SE01+NA2052-S1_PB" AND "01_PushButton"."SE01+NA1072-S1_PB" AND "01_PushButton"."SE01+NA2053-S1_PB" AND "01_PushButton"."SE01+NA2054-S1_PB" AND "01_PushButton"."SE01+NA2055-S1_PB" AND "01_PushButton"."SE01+NA2056-S1_PB" AND "01_PushButton"."SE01+NA1073-S1_PB" AND "01_PushButton"."SC00+UC254.VS019-9SF2_PB" AND "01_PushButton"."SE01+NA2045-S1_PB" AND "01_PushButton"."SE01+NA2046-S1_PB" AND "01_PushButton"."SE01+NA2047-S1_PB" AND "01_PushButton"."SE01+NA1062-S1_PB" AND "01_PushButton"."SE01+NA1063-S1_PB" AND "01_PushButton"."SE01+NA1064-S1_PB" AND "01_PushButton"."SE01+NA1065-S1_PB" AND "01_PushButton"."SE01+NA1066-S1_PB" AND "01_PushButton"."SE01+NA2044-S1_PB" AND "01_PushButton"."SC00+UC244.VS019-9SF2_PB" AND "01_PushButton"."SE01+NA2041-S1_PB" AND "01_PushButton"."SE01+NA2042-S1_PB" AND "01_PushButton"."SE01+NA2043-S1_PB" AND "01_PushButton"."SE01+NA1057-S1_PB" AND "01_PushButton"."SE01+NA1058-S1_PB" AND "01_PushButton"."SE01+NA1059-S1_PB" AND "01_PushButton"."SE01+NA1060-S1_PB" AND "01_PushButton"."SE01+NA1061-S1_PB" AND "01_PushButton"."SE01+NA2040-S1_PB" AND "01_PushButton"."SC00+UC234.VS019-9SF2_PB" AND "01_PushButton"."SE01+NA2037-S1_PB" AND "01_PushButton"."SE01+NA2038-S1_PB" AND "01_PushButton"."SE01+NA2039-S1_PB" AND "01_PushButton"."SE01+NA1116-S1_PB" AND "01_PushButton"."SE01+NA1051-S1_PB" AND "01_PushButton"."SE01+NA1053-S1_PB" AND "01_PushButton"."SE01+NA1054-S1_PB" AND "01_PushButton"."SE01+NA1055-S1_PB" AND "01_PushButton"."SE01+NA1056-S1_PB" AND "01_PushButton"."SE01+NA2036-S1_PB" AND "01_PushButton"."SE01+NA3025-S1_PB" AND "01_PushButton"."SE01+NA3026-S1_PB" AND "01_PushButton"."SC00+UC224.VS019-9SF2_PB" AND "01_PushButton"."SE01+NA2033-S1_PB" AND "01_PushButton"."SE01+NA2034-S1_PB" AND "01_PushButton"."SE01+NA2035-S1_PB" AND "01_PushButton"."SE01+NA1115-S1_PB" AND "01_PushButton"."SE01+NA1047-S1_PB" AND "01_PushButton"."SE01+NA1048-S1_PB" AND "01_PushButton"."SE01+NA1049-S1_PB" AND "01_PushButton"."SE01+NA1050-S1_PB" AND "01_PushButton"."SE01+NA1051-S1_PB" AND "01_PushButton"."SE01+NA2032-S1_PB" AND "01_PushButton"."SC00+UC214.VS019-9SF2_PB" AND "01_PushButton"."SE01+NA2029-S1_PB" AND "01_PushButton"."SE01+NA2030-S1_PB" AND "01_PushButton"."SE01+NA2031-S1_PB" AND "01_PushButton"."SE01+NA1041-S1_PB" AND "01_PushButton"."SE01+NA1042-S1_PB" AND "01_PushButton"."SE01+NA1043-S1_PB" AND "01_PushButton"."SE01+NA1044-S1_PB" AND "01_PushButton"."SE01+NA1045-S1_PB" AND "01_PushButton"."SE01+NA2028-S1_PB" AND "01_PushButton"."SE01+NA1114-S1_PB" AND "01_PushButton"."SE01+NA2075-S1_PB" AND "01_PushButton"."SE01+NA2077-S1_PB" AND "01_PushButton"."SE01+NA1113-S1_PB" AND "01_PushButton"."SE01+NA1112-S1_PB" AND "01_PushButton".FALSE AND "01_PushButton".FALSE AND "01_PushButton".FALSE AND "01_PushButton".FALSE AND "01_PushButton".FALSE AND "01_PushButton".FALSE AND "01_PushButton".FALSE AND "01_PushButton".FALSE AND "01_PushButton".FALSE AND "01_PushButton".FALSE AND "01_PushButton".FALSE AND "01_PushButton".FALSE AND "01_PushButton".FALSE AND "01_PushButton".FALSE AND "01_PushButton".FALSE AND "01_PushButton".FALSE AND "01_PushButton".FALSE AND "01_PushButton".FALSE AND "01_PushButton".FALSE AND "01_PushButton".FALSE AND "01_PushButton".FALSE AND "01_PushButton".FALSE AND "01_PushButton".FALSE AND "01_PushButton".FALSE AND "01_PushButton".FALSE AND "01_PushButton".FALSE AND "01_PushButton".FALSE AND "01_PushButton".FALSE AND "01_PushButton".FALSE AND "01_PushButton".FALSE AND "01_PushButton".FALSE AND "01_PushButton".FALSE AND "01_PushButton".FALSE AND "01_PushButton".FALSE AND "01_PushButton".FALSE AND "01_PushButton".FALSE AND "01_PushButton".FALSE AND "01_PushButton".FALSE AND "01_PushButton".FALSE AND "01_PushButton".FALSE AND "01_PushButton".FALSE AND "01_PushButton".FALSE AND "01_PushButton".FALSE AND "01_PushButton".FALSE AND "01_PushButton".FALSE AND "01_PushButton".FALSE AND "01_PushButton".FALSE AND "01_PushButton".FALSE AND "01_PushButton".FALSE AND "01_PushButton".FALSE AND "01_PushButton".FALSE AND "01_PushButton".FALSE AND "01_PushButton".FALSE AND "01_PushButton".FALSE;
END_REGION
END_FUNCTION

FUNCTION "04_ESTOP" : Void   // FC5, F_FBD
TITLE = EMERGENCY STOP
{ S7_Optimized_Access := 'TRUE' }
VERSION : 0.1
BEGIN

REGION Network 1: ^S1 | Sorter COY Upper [=SC01]
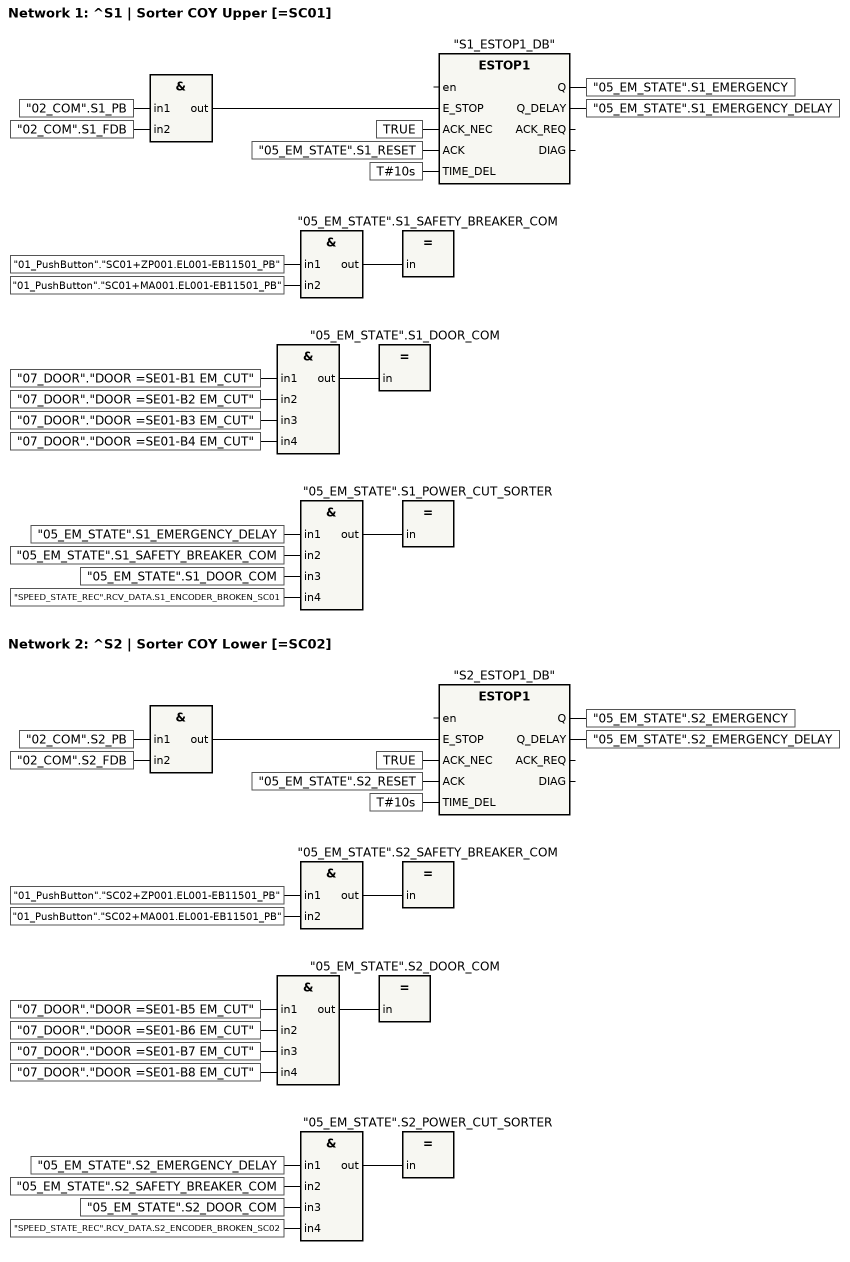
   "S1_ESTOP1_DB"(E_STOP := "02_COM".S1_PB AND "02_COM".S1_FDB,   // ESTOP1
                  ACK_NEC := TRUE,
                  ACK := "05_EM_STATE".S1_RESET,
                  TIME_DEL := T#10s,
                  Q => "05_EM_STATE".S1_EMERGENCY,
                  Q_DELAY => "05_EM_STATE".S1_EMERGENCY_DELAY);
   "05_EM_STATE".S1_SAFETY_BREAKER_COM := "01_PushButton"."SC01+ZP001.EL001-EB11501_PB" AND "01_PushButton"."SC01+MA001.EL001-EB11501_PB";
   "05_EM_STATE".S1_DOOR_COM := "07_DOOR"."DOOR =SE01-B1 EM_CUT" AND "07_DOOR"."DOOR =SE01-B2 EM_CUT" AND "07_DOOR"."DOOR =SE01-B3 EM_CUT" AND "07_DOOR"."DOOR =SE01-B4 EM_CUT";
   "05_EM_STATE".S1_POWER_CUT_SORTER := "05_EM_STATE".S1_EMERGENCY_DELAY AND "05_EM_STATE".S1_SAFETY_BREAKER_COM AND "05_EM_STATE".S1_DOOR_COM AND "SPEED_STATE_REC".RCV_DATA.S1_ENCODER_BROKEN_SC01;
END_REGION

REGION Network 2: ^S2 | Sorter COY Lower [=SC02]
   "S2_ESTOP1_DB"(E_STOP := "02_COM".S2_PB AND "02_COM".S2_FDB,   // ESTOP1
                  ACK_NEC := TRUE,
                  ACK := "05_EM_STATE".S2_RESET,
                  TIME_DEL := T#10s,
                  Q => "05_EM_STATE".S2_EMERGENCY,
                  Q_DELAY => "05_EM_STATE".S2_EMERGENCY_DELAY);
   "05_EM_STATE".S2_SAFETY_BREAKER_COM := "01_PushButton"."SC02+ZP001.EL001-EB11501_PB" AND "01_PushButton"."SC02+MA001.EL001-EB11501_PB";
   "05_EM_STATE".S2_DOOR_COM := "07_DOOR"."DOOR =SE01-B5 EM_CUT" AND "07_DOOR"."DOOR =SE01-B6 EM_CUT" AND "07_DOOR"."DOOR =SE01-B7 EM_CUT" AND "07_DOOR"."DOOR =SE01-B8 EM_CUT";
   "05_EM_STATE".S2_POWER_CUT_SORTER := "05_EM_STATE".S2_EMERGENCY_DELAY AND "05_EM_STATE".S2_SAFETY_BREAKER_COM AND "05_EM_STATE".S2_DOOR_COM AND "SPEED_STATE_REC".RCV_DATA.S2_ENCODER_BROKEN_SC02;
END_REGION

REGION Network 3: ^S3 | Sorter FLY Upper [=SF03]
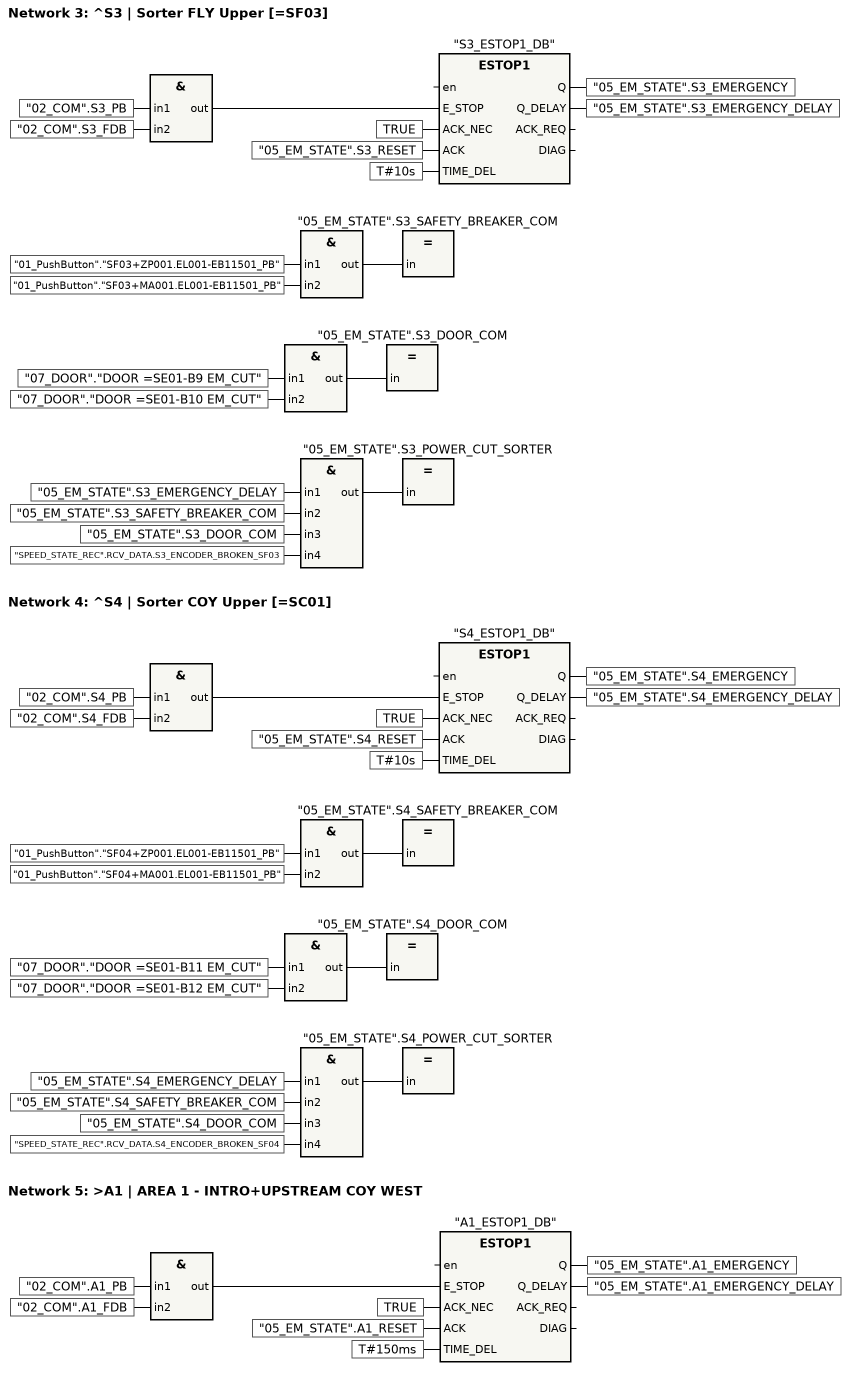
   "S3_ESTOP1_DB"(E_STOP := "02_COM".S3_PB AND "02_COM".S3_FDB,   // ESTOP1
                  ACK_NEC := TRUE,
                  ACK := "05_EM_STATE".S3_RESET,
                  TIME_DEL := T#10s,
                  Q => "05_EM_STATE".S3_EMERGENCY,
                  Q_DELAY => "05_EM_STATE".S3_EMERGENCY_DELAY);
   "05_EM_STATE".S3_SAFETY_BREAKER_COM := "01_PushButton"."SF03+ZP001.EL001-EB11501_PB" AND "01_PushButton"."SF03+MA001.EL001-EB11501_PB";
   "05_EM_STATE".S3_DOOR_COM := "07_DOOR"."DOOR =SE01-B9 EM_CUT" AND "07_DOOR"."DOOR =SE01-B10 EM_CUT";
   "05_EM_STATE".S3_POWER_CUT_SORTER := "05_EM_STATE".S3_EMERGENCY_DELAY AND "05_EM_STATE".S3_SAFETY_BREAKER_COM AND "05_EM_STATE".S3_DOOR_COM AND "SPEED_STATE_REC".RCV_DATA.S3_ENCODER_BROKEN_SF03;
END_REGION

REGION Network 4: ^S4 | Sorter COY Upper [=SC01]
   "S4_ESTOP1_DB"(E_STOP := "02_COM".S4_PB AND "02_COM".S4_FDB,   // ESTOP1
                  ACK_NEC := TRUE,
                  ACK := "05_EM_STATE".S4_RESET,
                  TIME_DEL := T#10s,
                  Q => "05_EM_STATE".S4_EMERGENCY,
                  Q_DELAY => "05_EM_STATE".S4_EMERGENCY_DELAY);
   "05_EM_STATE".S4_SAFETY_BREAKER_COM := "01_PushButton"."SF04+ZP001.EL001-EB11501_PB" AND "01_PushButton"."SF04+MA001.EL001-EB11501_PB";
   "05_EM_STATE".S4_DOOR_COM := "07_DOOR"."DOOR =SE01-B11 EM_CUT" AND "07_DOOR"."DOOR =SE01-B12 EM_CUT";
   "05_EM_STATE".S4_POWER_CUT_SORTER := "05_EM_STATE".S4_EMERGENCY_DELAY AND "05_EM_STATE".S4_SAFETY_BREAKER_COM AND "05_EM_STATE".S4_DOOR_COM AND "SPEED_STATE_REC".RCV_DATA.S4_ENCODER_BROKEN_SF04;
END_REGION

REGION Network 5: >A1 | AREA 1 - INTRO+UPSTREAM COY WEST
   "A1_ESTOP1_DB"(E_STOP := "02_COM".A1_PB AND "02_COM".A1_FDB,   // ESTOP1
                  ACK_NEC := TRUE,
                  ACK := "05_EM_STATE".A1_RESET,
                  TIME_DEL := T#150ms,
                  Q => "05_EM_STATE".A1_EMERGENCY,
                  Q_DELAY => "05_EM_STATE".A1_EMERGENCY_DELAY);
END_REGION

REGION Network 6: >A2 | AREA 2 - UPSTREAM FLY WEST 5FSN_115/117
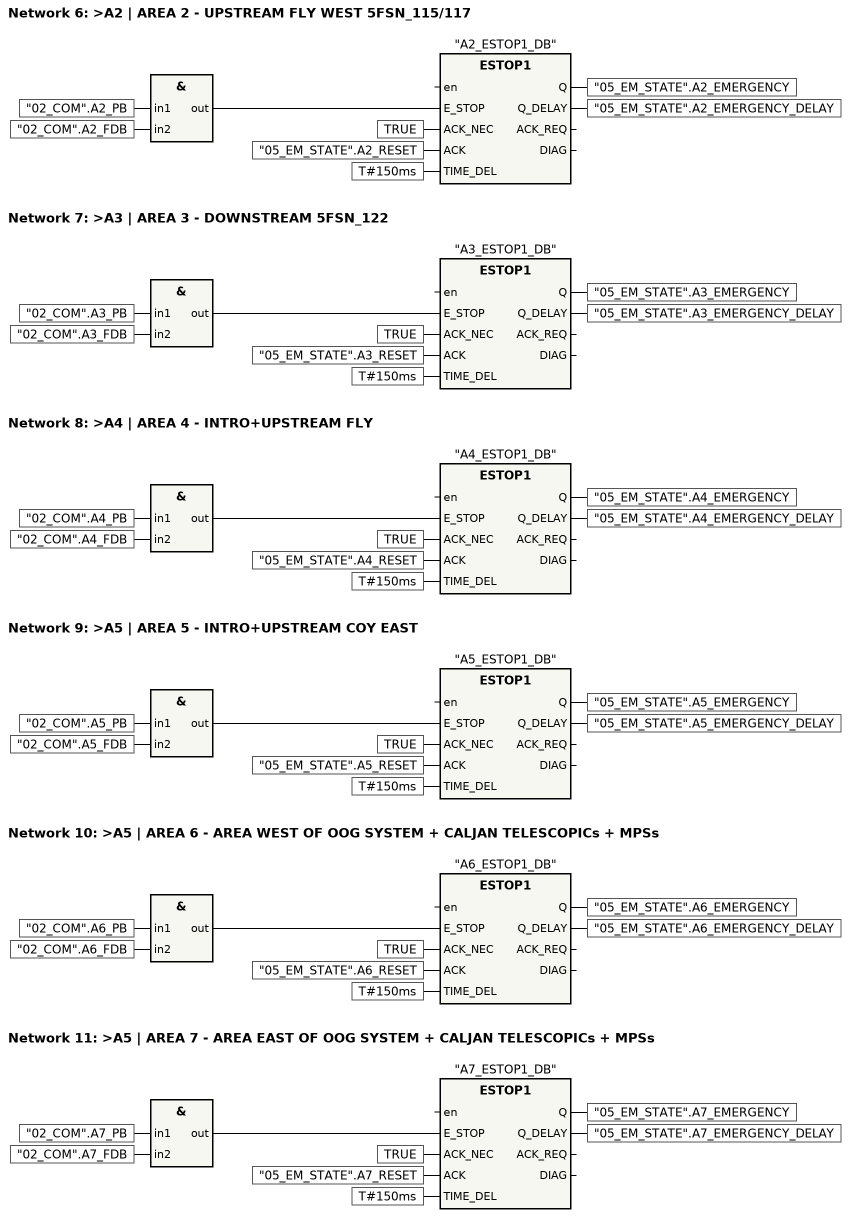
   "A2_ESTOP1_DB"(E_STOP := "02_COM".A2_PB AND "02_COM".A2_FDB,   // ESTOP1
                  ACK_NEC := TRUE,
                  ACK := "05_EM_STATE".A2_RESET,
                  TIME_DEL := T#150ms,
                  Q => "05_EM_STATE".A2_EMERGENCY,
                  Q_DELAY => "05_EM_STATE".A2_EMERGENCY_DELAY);
END_REGION

REGION Network 7: >A3 | AREA 3 - DOWNSTREAM 5FSN_122
   "A3_ESTOP1_DB"(E_STOP := "02_COM".A3_PB AND "02_COM".A3_FDB,   // ESTOP1
                  ACK_NEC := TRUE,
                  ACK := "05_EM_STATE".A3_RESET,
                  TIME_DEL := T#150ms,
                  Q => "05_EM_STATE".A3_EMERGENCY,
                  Q_DELAY => "05_EM_STATE".A3_EMERGENCY_DELAY);
END_REGION

REGION Network 8: >A4 | AREA 4 - INTRO+UPSTREAM FLY
   "A4_ESTOP1_DB"(E_STOP := "02_COM".A4_PB AND "02_COM".A4_FDB,   // ESTOP1
                  ACK_NEC := TRUE,
                  ACK := "05_EM_STATE".A4_RESET,
                  TIME_DEL := T#150ms,
                  Q => "05_EM_STATE".A4_EMERGENCY,
                  Q_DELAY => "05_EM_STATE".A4_EMERGENCY_DELAY);
END_REGION

REGION Network 9: >A5 | AREA 5 - INTRO+UPSTREAM COY EAST
   "A5_ESTOP1_DB"(E_STOP := "02_COM".A5_PB AND "02_COM".A5_FDB,   // ESTOP1
                  ACK_NEC := TRUE,
                  ACK := "05_EM_STATE".A5_RESET,
                  TIME_DEL := T#150ms,
                  Q => "05_EM_STATE".A5_EMERGENCY,
                  Q_DELAY => "05_EM_STATE".A5_EMERGENCY_DELAY);
END_REGION

REGION Network 10: >A5 | AREA 6 - AREA WEST OF OOG SYSTEM + CALJAN TELESCOPICs + MPSs
   "A6_ESTOP1_DB"(E_STOP := "02_COM".A6_PB AND "02_COM".A6_FDB,   // ESTOP1
                  ACK_NEC := TRUE,
                  ACK := "05_EM_STATE".A6_RESET,
                  TIME_DEL := T#150ms,
                  Q => "05_EM_STATE".A6_EMERGENCY,
                  Q_DELAY => "05_EM_STATE".A6_EMERGENCY_DELAY);
END_REGION

REGION Network 11: >A5 | AREA 7 - AREA EAST OF OOG SYSTEM + CALJAN TELESCOPICs + MPSs
   "A7_ESTOP1_DB"(E_STOP := "02_COM".A7_PB AND "02_COM".A7_FDB,   // ESTOP1
                  ACK_NEC := TRUE,
                  ACK := "05_EM_STATE".A7_RESET,
                  TIME_DEL := T#150ms,
                  Q => "05_EM_STATE".A7_EMERGENCY,
                  Q_DELAY => "05_EM_STATE".A7_EMERGENCY_DELAY);
END_REGION

REGION Network 12: #L1 Local C&E - Cause: Door =SC00+UC114.VS019-8AF3 (I2172.3) / Effect: =SC00+UC114.VS019
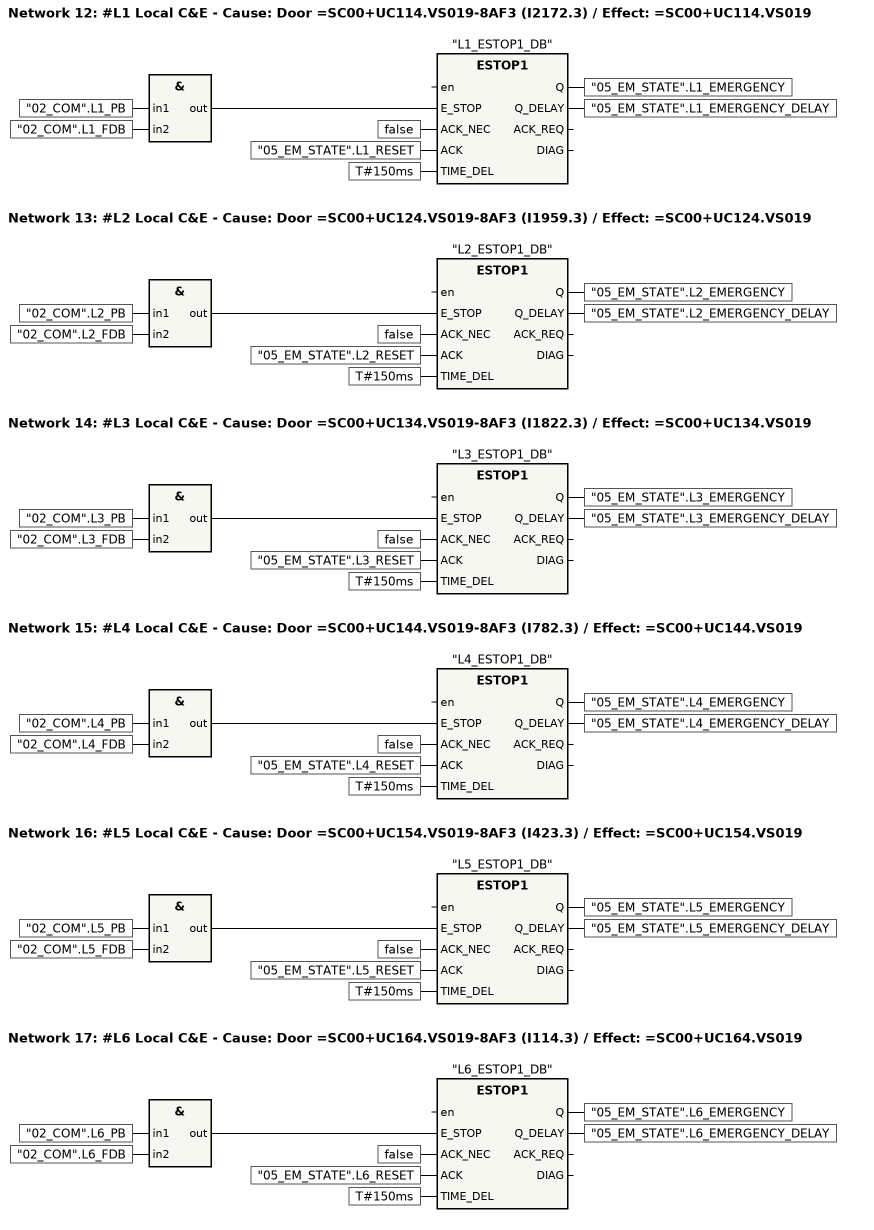
   "L1_ESTOP1_DB"(E_STOP := "02_COM".L1_PB AND "02_COM".L1_FDB,   // ESTOP1
                  ACK_NEC := false,
                  ACK := "05_EM_STATE".L1_RESET,
                  TIME_DEL := T#150ms,
                  Q => "05_EM_STATE".L1_EMERGENCY,
                  Q_DELAY => "05_EM_STATE".L1_EMERGENCY_DELAY);
END_REGION

REGION Network 13: #L2 Local C&E - Cause: Door =SC00+UC124.VS019-8AF3 (I1959.3) / Effect: =SC00+UC124.VS019
   "L2_ESTOP1_DB"(E_STOP := "02_COM".L2_PB AND "02_COM".L2_FDB,   // ESTOP1
                  ACK_NEC := false,
                  ACK := "05_EM_STATE".L2_RESET,
                  TIME_DEL := T#150ms,
                  Q => "05_EM_STATE".L2_EMERGENCY,
                  Q_DELAY => "05_EM_STATE".L2_EMERGENCY_DELAY);
END_REGION

REGION Network 14: #L3 Local C&E - Cause: Door =SC00+UC134.VS019-8AF3 (I1822.3) / Effect: =SC00+UC134.VS019
   "L3_ESTOP1_DB"(E_STOP := "02_COM".L3_PB AND "02_COM".L3_FDB,   // ESTOP1
                  ACK_NEC := false,
                  ACK := "05_EM_STATE".L3_RESET,
                  TIME_DEL := T#150ms,
                  Q => "05_EM_STATE".L3_EMERGENCY,
                  Q_DELAY => "05_EM_STATE".L3_EMERGENCY_DELAY);
END_REGION

REGION Network 15: #L4 Local C&E - Cause: Door =SC00+UC144.VS019-8AF3 (I782.3) / Effect: =SC00+UC144.VS019
   "L4_ESTOP1_DB"(E_STOP := "02_COM".L4_PB AND "02_COM".L4_FDB,   // ESTOP1
                  ACK_NEC := false,
                  ACK := "05_EM_STATE".L4_RESET,
                  TIME_DEL := T#150ms,
                  Q => "05_EM_STATE".L4_EMERGENCY,
                  Q_DELAY => "05_EM_STATE".L4_EMERGENCY_DELAY);
END_REGION

REGION Network 16: #L5 Local C&E - Cause: Door =SC00+UC154.VS019-8AF3 (I423.3) / Effect: =SC00+UC154.VS019
   "L5_ESTOP1_DB"(E_STOP := "02_COM".L5_PB AND "02_COM".L5_FDB,   // ESTOP1
                  ACK_NEC := false,
                  ACK := "05_EM_STATE".L5_RESET,
                  TIME_DEL := T#150ms,
                  Q => "05_EM_STATE".L5_EMERGENCY,
                  Q_DELAY => "05_EM_STATE".L5_EMERGENCY_DELAY);
END_REGION

REGION Network 17: #L6 Local C&E - Cause: Door =SC00+UC164.VS019-8AF3 (I114.3) / Effect: =SC00+UC164.VS019
   "L6_ESTOP1_DB"(E_STOP := "02_COM".L6_PB AND "02_COM".L6_FDB,   // ESTOP1
                  ACK_NEC := false,
                  ACK := "05_EM_STATE".L6_RESET,
                  TIME_DEL := T#150ms,
                  Q => "05_EM_STATE".L6_EMERGENCY,
                  Q_DELAY => "05_EM_STATE".L6_EMERGENCY_DELAY);
END_REGION

REGION Network 18: #L7 Local C&E - Cause: Door =SC00+UC175.VS019-8AF3 (I2461.1) / Effect: =SC00+UC175.VS019
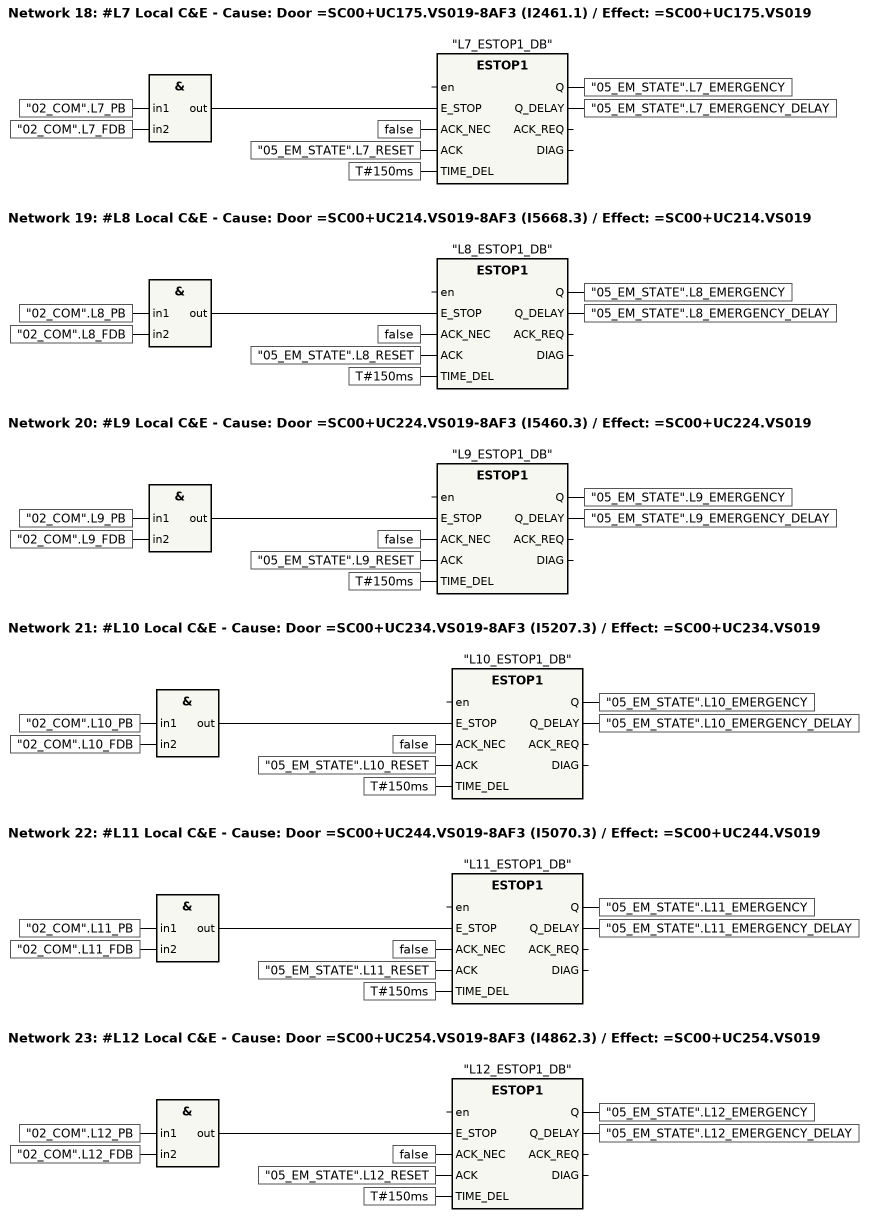
   "L7_ESTOP1_DB"(E_STOP := "02_COM".L7_PB AND "02_COM".L7_FDB,   // ESTOP1
                  ACK_NEC := false,
                  ACK := "05_EM_STATE".L7_RESET,
                  TIME_DEL := T#150ms,
                  Q => "05_EM_STATE".L7_EMERGENCY,
                  Q_DELAY => "05_EM_STATE".L7_EMERGENCY_DELAY);
END_REGION

REGION Network 19: #L8 Local C&E - Cause: Door =SC00+UC214.VS019-8AF3 (I5668.3) / Effect: =SC00+UC214.VS019
   "L8_ESTOP1_DB"(E_STOP := "02_COM".L8_PB AND "02_COM".L8_FDB,   // ESTOP1
                  ACK_NEC := false,
                  ACK := "05_EM_STATE".L8_RESET,
                  TIME_DEL := T#150ms,
                  Q => "05_EM_STATE".L8_EMERGENCY,
                  Q_DELAY => "05_EM_STATE".L8_EMERGENCY_DELAY);
END_REGION

REGION Network 20: #L9 Local C&E - Cause: Door =SC00+UC224.VS019-8AF3 (I5460.3) / Effect: =SC00+UC224.VS019
   "L9_ESTOP1_DB"(E_STOP := "02_COM".L9_PB AND "02_COM".L9_FDB,   // ESTOP1
                  ACK_NEC := false,
                  ACK := "05_EM_STATE".L9_RESET,
                  TIME_DEL := T#150ms,
                  Q => "05_EM_STATE".L9_EMERGENCY,
                  Q_DELAY => "05_EM_STATE".L9_EMERGENCY_DELAY);
END_REGION

REGION Network 21: #L10 Local C&E - Cause: Door =SC00+UC234.VS019-8AF3 (I5207.3) / Effect: =SC00+UC234.VS019
   "L10_ESTOP1_DB"(E_STOP := "02_COM".L10_PB AND "02_COM".L10_FDB,   // ESTOP1
                   ACK_NEC := false,
                   ACK := "05_EM_STATE".L10_RESET,
                   TIME_DEL := T#150ms,
                   Q => "05_EM_STATE".L10_EMERGENCY,
                   Q_DELAY => "05_EM_STATE".L10_EMERGENCY_DELAY);
END_REGION

REGION Network 22: #L11 Local C&E - Cause: Door =SC00+UC244.VS019-8AF3 (I5070.3) / Effect: =SC00+UC244.VS019
   "L11_ESTOP1_DB"(E_STOP := "02_COM".L11_PB AND "02_COM".L11_FDB,   // ESTOP1
                   ACK_NEC := false,
                   ACK := "05_EM_STATE".L11_RESET,
                   TIME_DEL := T#150ms,
                   Q => "05_EM_STATE".L11_EMERGENCY,
                   Q_DELAY => "05_EM_STATE".L11_EMERGENCY_DELAY);
END_REGION

REGION Network 23: #L12 Local C&E - Cause: Door =SC00+UC254.VS019-8AF3 (I4862.3) / Effect: =SC00+UC254.VS019
   "L12_ESTOP1_DB"(E_STOP := "02_COM".L12_PB AND "02_COM".L12_FDB,   // ESTOP1
                   ACK_NEC := false,
                   ACK := "05_EM_STATE".L12_RESET,
                   TIME_DEL := T#150ms,
                   Q => "05_EM_STATE".L12_EMERGENCY,
                   Q_DELAY => "05_EM_STATE".L12_EMERGENCY_DELAY);
END_REGION

REGION Network 24: #L13 Local C&E - Cause: Door =SC00+UC264.VS019-8AF3 (I4423.3) / Effect: =SC00+UC264.VS019
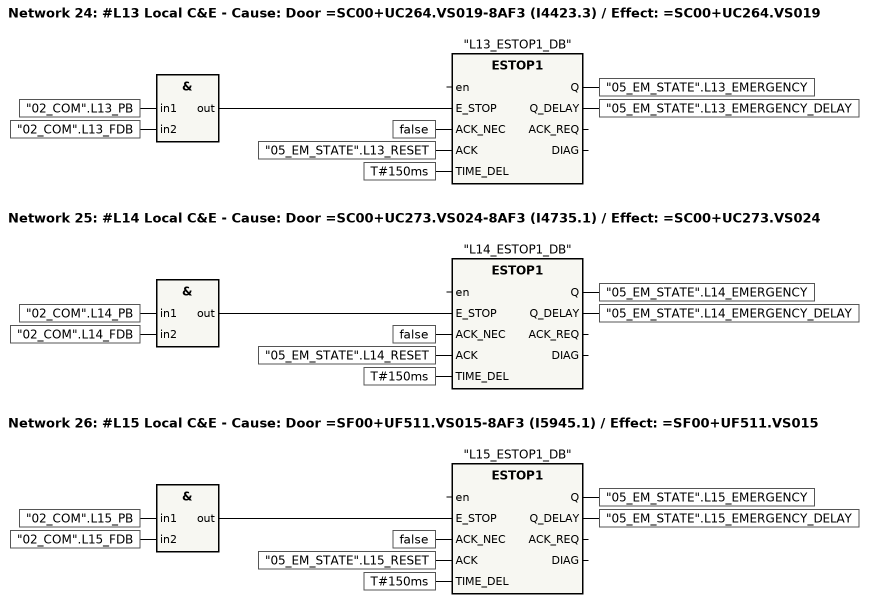
   "L13_ESTOP1_DB"(E_STOP := "02_COM".L13_PB AND "02_COM".L13_FDB,   // ESTOP1
                   ACK_NEC := false,
                   ACK := "05_EM_STATE".L13_RESET,
                   TIME_DEL := T#150ms,
                   Q => "05_EM_STATE".L13_EMERGENCY,
                   Q_DELAY => "05_EM_STATE".L13_EMERGENCY_DELAY);
END_REGION

REGION Network 25: #L14 Local C&E - Cause: Door =SC00+UC273.VS024-8AF3 (I4735.1) / Effect: =SC00+UC273.VS024
   "L14_ESTOP1_DB"(E_STOP := "02_COM".L14_PB AND "02_COM".L14_FDB,   // ESTOP1
                   ACK_NEC := false,
                   ACK := "05_EM_STATE".L14_RESET,
                   TIME_DEL := T#150ms,
                   Q => "05_EM_STATE".L14_EMERGENCY,
                   Q_DELAY => "05_EM_STATE".L14_EMERGENCY_DELAY);
END_REGION

REGION Network 26: #L15 Local C&E - Cause: Door =SF00+UF511.VS015-8AF3 (I5945.1) / Effect: =SF00+UF511.VS015
   "L15_ESTOP1_DB"(E_STOP := "02_COM".L15_PB AND "02_COM".L15_FDB,   // ESTOP1
                   ACK_NEC := false,
                   ACK := "05_EM_STATE".L15_RESET,
                   TIME_DEL := T#150ms,
                   Q => "05_EM_STATE".L15_EMERGENCY,
                   Q_DELAY => "05_EM_STATE".L15_EMERGENCY_DELAY);
END_REGION
END_FUNCTION

FUNCTION "05_Output Feedback" : Void   // FC6, F_FBD
TITLE = Manage Safety Outputs
{ S7_Optimized_Access := 'TRUE' }
VERSION : 0.1
   VAR_TEMP
      DU_EX : Bool;
      ISPC_EX : Bool;
      ZONE_EX : Bool;
   END_VAR
BEGIN

REGION Network 1: Area S1 =SC01+DU001/DU019.EL001 DRIVE UNIT DU001/DU019
   // "=SC01+LV001.EL001-Q32002 ( =SC01+DU001/DU018/DU019.EL001)"
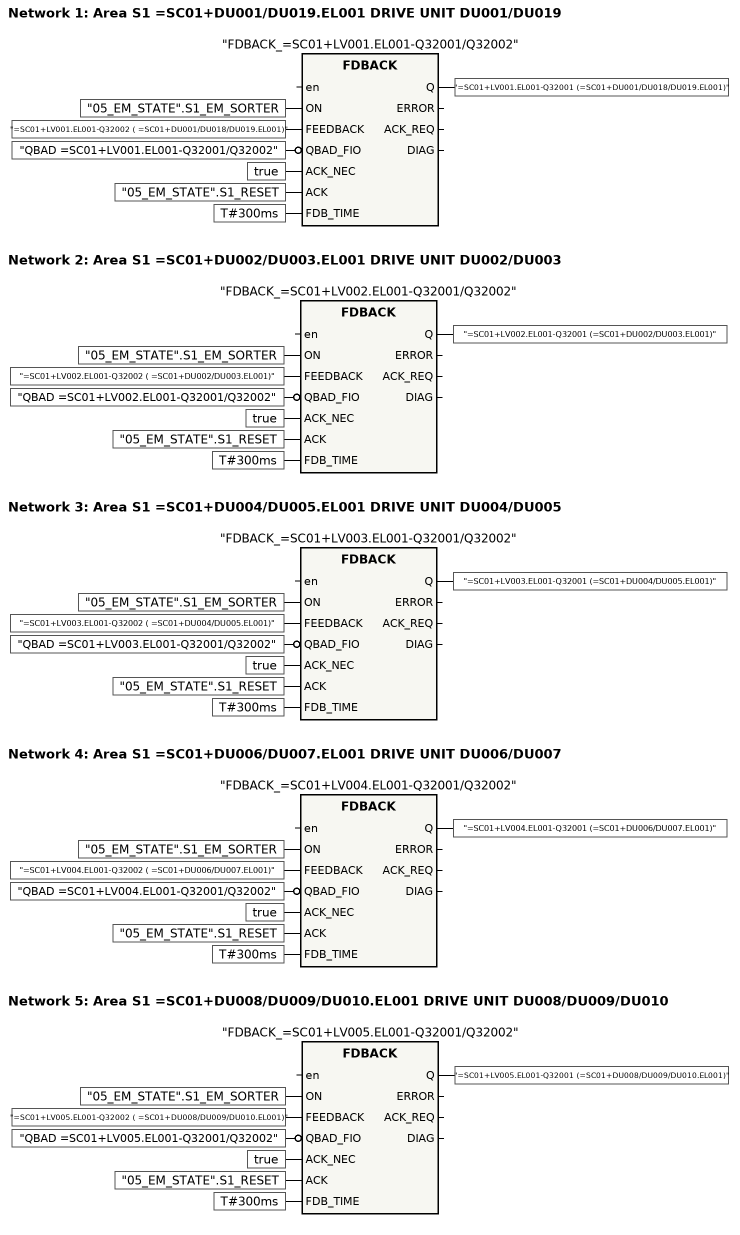
   "FDBACK_=SC01+LV001.EL001-Q32001/Q32002"(ON := "05_EM_STATE".S1_EM_SORTER,   // FDBACK
                           FEEDBACK := "=SC01+LV001.EL001-Q32002 ( =SC01+DU001/DU018/DU019.EL001)",
                           QBAD_FIO := NOT "QBAD =SC01+LV001.EL001-Q32001/Q32002",
                           ACK_NEC := true,
                           ACK := "05_EM_STATE".S1_RESET,
                           FDB_TIME := T#300ms,
                           Q => "=SC01+LV001.EL001-Q32001 (=SC01+DU001/DU018/DU019.EL001)");
END_REGION

REGION Network 2: Area S1 =SC01+DU002/DU003.EL001 DRIVE UNIT DU002/DU003
   "FDBACK_=SC01+LV002.EL001-Q32001/Q32002"(ON := "05_EM_STATE".S1_EM_SORTER,   // FDBACK
                           FEEDBACK := "=SC01+LV002.EL001-Q32002 ( =SC01+DU002/DU003.EL001)",
                           QBAD_FIO := NOT "QBAD =SC01+LV002.EL001-Q32001/Q32002",
                           ACK_NEC := true,
                           ACK := "05_EM_STATE".S1_RESET,
                           FDB_TIME := T#300ms,
                           Q => "=SC01+LV002.EL001-Q32001 (=SC01+DU002/DU003.EL001)");
END_REGION

REGION Network 3: Area S1 =SC01+DU004/DU005.EL001 DRIVE UNIT DU004/DU005
   "FDBACK_=SC01+LV003.EL001-Q32001/Q32002"(ON := "05_EM_STATE".S1_EM_SORTER,   // FDBACK
                           FEEDBACK := "=SC01+LV003.EL001-Q32002 ( =SC01+DU004/DU005.EL001)",
                           QBAD_FIO := NOT "QBAD =SC01+LV003.EL001-Q32001/Q32002",
                           ACK_NEC := true,
                           ACK := "05_EM_STATE".S1_RESET,
                           FDB_TIME := T#300ms,
                           Q => "=SC01+LV003.EL001-Q32001 (=SC01+DU004/DU005.EL001)");
END_REGION

REGION Network 4: Area S1 =SC01+DU006/DU007.EL001 DRIVE UNIT DU006/DU007
   "FDBACK_=SC01+LV004.EL001-Q32001/Q32002"(ON := "05_EM_STATE".S1_EM_SORTER,   // FDBACK
                           FEEDBACK := "=SC01+LV004.EL001-Q32002 ( =SC01+DU006/DU007.EL001)",
                           QBAD_FIO := NOT "QBAD =SC01+LV004.EL001-Q32001/Q32002",
                           ACK_NEC := true,
                           ACK := "05_EM_STATE".S1_RESET,
                           FDB_TIME := T#300ms,
                           Q => "=SC01+LV004.EL001-Q32001 (=SC01+DU006/DU007.EL001)");
END_REGION

REGION Network 5: Area S1 =SC01+DU008/DU009/DU010.EL001 DRIVE UNIT DU008/DU009/DU010
   "FDBACK_=SC01+LV005.EL001-Q32001/Q32002"(ON := "05_EM_STATE".S1_EM_SORTER,   // FDBACK
                           FEEDBACK := "=SC01+LV005.EL001-Q32002 ( =SC01+DU008/DU009/DU010.EL001)",
                           QBAD_FIO := NOT "QBAD =SC01+LV005.EL001-Q32001/Q32002",
                           ACK_NEC := true,
                           ACK := "05_EM_STATE".S1_RESET,
                           FDB_TIME := T#300ms,
                           Q => "=SC01+LV005.EL001-Q32001 (=SC01+DU008/DU009/DU010.EL001)");
END_REGION

REGION Network 6: Area S1 =SC01+DU011/DU012/DU013.EL001 DRIVE UNIT DU011/DU012/DU013
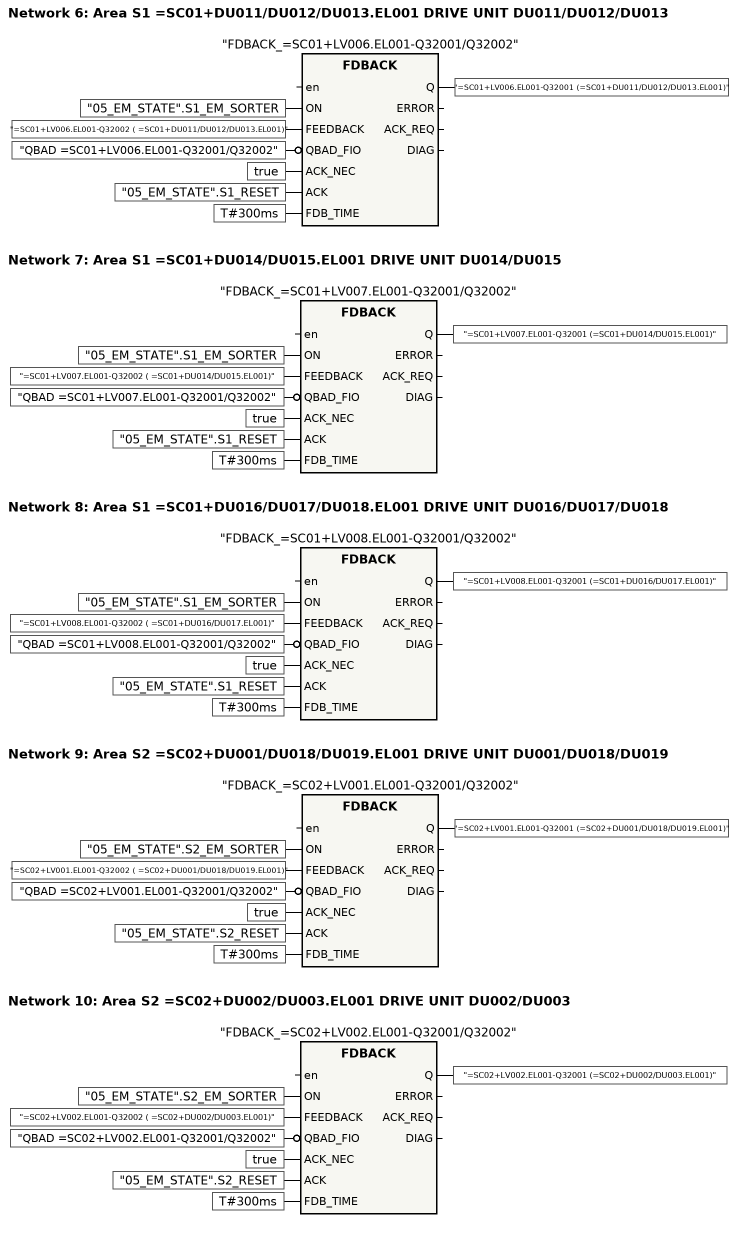
   "FDBACK_=SC01+LV006.EL001-Q32001/Q32002"(ON := "05_EM_STATE".S1_EM_SORTER,   // FDBACK
                           FEEDBACK := "=SC01+LV006.EL001-Q32002 ( =SC01+DU011/DU012/DU013.EL001)",
                           QBAD_FIO := NOT "QBAD =SC01+LV006.EL001-Q32001/Q32002",
                           ACK_NEC := true,
                           ACK := "05_EM_STATE".S1_RESET,
                           FDB_TIME := T#300ms,
                           Q => "=SC01+LV006.EL001-Q32001 (=SC01+DU011/DU012/DU013.EL001)");
END_REGION

REGION Network 7: Area S1 =SC01+DU014/DU015.EL001 DRIVE UNIT DU014/DU015
   "FDBACK_=SC01+LV007.EL001-Q32001/Q32002"(ON := "05_EM_STATE".S1_EM_SORTER,   // FDBACK
                           FEEDBACK := "=SC01+LV007.EL001-Q32002 ( =SC01+DU014/DU015.EL001)",
                           QBAD_FIO := NOT "QBAD =SC01+LV007.EL001-Q32001/Q32002",
                           ACK_NEC := true,
                           ACK := "05_EM_STATE".S1_RESET,
                           FDB_TIME := T#300ms,
                           Q => "=SC01+LV007.EL001-Q32001 (=SC01+DU014/DU015.EL001)");
END_REGION

REGION Network 8: Area S1 =SC01+DU016/DU017/DU018.EL001 DRIVE UNIT DU016/DU017/DU018
   "FDBACK_=SC01+LV008.EL001-Q32001/Q32002"(ON := "05_EM_STATE".S1_EM_SORTER,   // FDBACK
                           FEEDBACK := "=SC01+LV008.EL001-Q32002 ( =SC01+DU016/DU017.EL001)",
                           QBAD_FIO := NOT "QBAD =SC01+LV008.EL001-Q32001/Q32002",
                           ACK_NEC := true,
                           ACK := "05_EM_STATE".S1_RESET,
                           FDB_TIME := T#300ms,
                           Q => "=SC01+LV008.EL001-Q32001 (=SC01+DU016/DU017.EL001)");
END_REGION

REGION Network 9: Area S2 =SC02+DU001/DU018/DU019.EL001 DRIVE UNIT DU001/DU018/DU019
   "FDBACK_=SC02+LV001.EL001-Q32001/Q32002"(ON := "05_EM_STATE".S2_EM_SORTER,   // FDBACK
                           FEEDBACK := "=SC02+LV001.EL001-Q32002 ( =SC02+DU001/DU018/DU019.EL001)",
                           QBAD_FIO := NOT "QBAD =SC02+LV001.EL001-Q32001/Q32002",
                           ACK_NEC := true,
                           ACK := "05_EM_STATE".S2_RESET,
                           FDB_TIME := T#300ms,
                           Q => "=SC02+LV001.EL001-Q32001 (=SC02+DU001/DU018/DU019.EL001)");
END_REGION

REGION Network 10: Area S2 =SC02+DU002/DU003.EL001 DRIVE UNIT DU002/DU003
   "FDBACK_=SC02+LV002.EL001-Q32001/Q32002"(ON := "05_EM_STATE".S2_EM_SORTER,   // FDBACK
                           FEEDBACK := "=SC02+LV002.EL001-Q32002 ( =SC02+DU002/DU003.EL001)",
                           QBAD_FIO := NOT "QBAD =SC02+LV002.EL001-Q32001/Q32002",
                           ACK_NEC := true,
                           ACK := "05_EM_STATE".S2_RESET,
                           FDB_TIME := T#300ms,
                           Q => "=SC02+LV002.EL001-Q32001 (=SC02+DU002/DU003.EL001)");
END_REGION

REGION Network 11: Area S2 =SC02+DU004/DU005.EL001 DRIVE UNIT DU004/DU005
